LIN {X 0,Y 524.534,Z 584.102,A -85,B 0,C 180,E1 -4783.363,E2 -4783.363} C_VEL
LIN {X 0,Y 524.942,Z 571.861,A -85,B 0,C 180,E1 -4784.637,E2 -4784.637} C_VEL
LIN {X 0,Y 525.437,Z 560.491,A -85,B 0,C 180,E1 -4785.626,E2 -4785.626} C_VEL
LIN {X 0,Y 525.876,Z 547.102,A -85,B 0,C 180,E1 -4786.598,E2 -4786.598} C_VEL
LIN {X 0,Y 526.385,Z 533.833,A -85,B 0,C 180,E1 -4787.382,E2 -4787.382} C_VEL
LIN {X 0,Y 526.784,Z 519.311,A -85,B 0,C 180,E1 -4788.07,E2 -4788.07} C_VEL
LIN {X 0,Y 527.168,Z 504.263,A -85,B 0,C 180,E1 -4788.61,E2 -4788.61} C_VEL
LIN {X 0,Y 527.486,Z 489.588,A -85,B 0,C 180,E1 -4788.979,E2 -4788.979} C_VEL
LIN {X 0,Y 527.689,Z 461.99,A -85,B 0,C 180,E1 -4789.4,E2 -4789.4} C_VEL
LIN {X 0,Y 528.491,Z 335.003,A -85,B 0,C 180,E1 -4791.175,E2 -4791.175} C_VEL
LIN {X 0,Y 525.773,Z 320.948,A -85,B 0,C 180,E1 -4791.508,E2 -4791.508} C_VEL
LIN {X 0,Y 526.419,Z 300.055,A -85,B 0,C 180,E1 -4794.238,E2 -4794.238} C_VEL
LIN {X 0,Y 526.82,Z 285.888,A -85,B 0,C 180,E1 -4796.119,E2 -4796.119} C_VEL
LIN {X 0,Y 524.339,Z 274.589,A -85,B 0,C 180,E1 -4797.793,E2 -4797.793} C_VEL
LIN {X 0,Y 523.945,Z 272.841,A -85,B 0,C 180,E1 -4798.082,E2 -4798.082} C_VEL
LIN {X 0,Y 523.94,Z 272.844,A -85,B 0,C 180,E1 -4800.853,E2 -4800.853} C_VEL
LIN {X 0,Y 523.926,Z 272.849,A -85,B 0,C 180,E1 -4803.728,E2 -4803.728} C_VEL
LIN {X 0,Y 523.887,Z 272.856,A -85,B 0,C 180,E1 -4806.398,E2 -4806.398} C_VEL
LIN {X 0,Y 523.911,Z 272.847,A -85,B 0,C 180,E1 -4809.085,E2 -4809.085} C_VEL
LIN {X 0,Y 523.898,Z 272.854,A -85,B 0,C 180,E1 -4812.124,E2 -4812.124} C_VEL
LIN {X 0,Y 523.934,Z 272.843,A -85,B 0,C 180,E1 -4815.31,E2 -4815.31} C_VEL
LIN {X 0,Y 523.92,Z 272.846,A -85,B 0,C 180,E1 -4818.693,E2 -4818.693} C_VEL
LIN {X 0,Y 523.898,Z 272.853,A -85,B 0,C 180,E1 -4821.896,E2 -4821.896} C_VEL
LIN {X 0,Y 523.911,Z 272.843,A -85,B 0,C 180,E1 -4824.912,E2 -4824.912} C_VEL
LIN {X 0,Y 523.932,Z 272.847,A -85,B 0,C 180,E1 -4827.679,E2 -4827.679} C_VEL
LIN {X 0,Y 523.948,Z 272.84,A -85,B 0,C 180,E1 -4830.676,E2 -4830.676} C_VEL
LIN {X 0,Y 523.887,Z 272.854,A -85,B 0,C 180,E1 -4833.723,E2 -4833.723} C_VEL
LIN {X 0,Y 523.904,Z 272.848,A -85,B 0,C 180,E1 -4836.268,E2 -4836.268} C_VEL
LIN {X 0,Y 523.94,Z 272.842,A -85,B 0,C 180,E1 -4838.765,E2 -4838.765} C_VEL
LIN {X 0,Y 523.928,Z 272.844,A -85,B 0,C 180,E1 -4841.219,E2 -4841.219} C_VEL
LIN {X 0,Y 523.898,Z 272.855,A -85,B 0,C 180,E1 -4843.637,E2 -4843.637} C_VEL
LIN {X 0,Y 523.921,Z 272.84,A -85,B 0,C 180,E1 -4846.026,E2 -4846.026} C_VEL
LIN {X 0,Y 523.955,Z 272.834,A -85,B 0,C 180,E1 -4848.392,E2 -4848.392} C_VEL
LIN {X 0,Y 523.937,Z 272.848,A -85,B 0,C 180,E1 -4851.514,E2 -4851.514} C_VEL
LIN {X 0,Y 524.026,Z 272.827,A -85,B 0,C 180,E1 -4854.612,E2 -4854.612} C_VEL
LIN {X 0,Y 524.088,Z 272.823,A -85,B 0,C 180,E1 -4857.693,E2 -4857.693} C_VEL
LIN {X 0,Y 524.078,Z 272.826,A -85,B 0,C 180,E1 -4859.999,E2 -4859.999} C_VEL
LIN {X 0,Y 524.02,Z 272.834,A -85,B 0,C 180,E1 -4863.074,E2 -4863.074} C_VEL
LIN {X 0,Y 523.975,Z 272.827,A -85,B 0,C 180,E1 -4866.158,E2 -4866.158} C_VEL
LIN {X 0,Y 523.929,Z 272.844,A -85,B 0,C 180,E1 -4869.262,E2 -4869.262} C_VEL
LIN {X 0,Y 523.983,Z 272.84,A -85,B 0,C 180,E1 -4871.733,E2 -4871.733} C_VEL
LIN {X 0,Y 523.97,Z 272.838,A -85,B 0,C 180,E1 -4875.046,E2 -4875.046} C_VEL
LIN {X 0,Y 523.901,Z 272.841,A -85,B 0,C 180,E1 -4877.97,E2 -4877.97} C_VEL
LIN {X 0,Y 523.938,Z 272.84,A -85,B 0,C 180,E1 -4880.41,E2 -4880.41} C_VEL
LIN {X 0,Y 523.892,Z 272.85,A -85,B 0,C 180,E1 -4882.893,E2 -4882.893} C_VEL
LIN {X 0,Y 523.886,Z 272.847,A -85,B 0,C 180,E1 -4885.42,E2 -4885.42} C_VEL
LIN {X 0,Y 523.891,Z 272.841,A -85,B 0,C 180,E1 -4888.001,E2 -4888.001} C_VEL
LIN {X 0,Y 523.919,Z 272.846,A -85,B 0,C 180,E1 -4890.851,E2 -4890.851} C_VEL
LIN {X 0,Y 523.91,Z 272.844,A -85,B 0,C 180,E1 -4893.728,E2 -4893.728} C_VEL
LIN {X 0,Y 523.881,Z 272.841,A -85,B 0,C 180,E1 -4896.399,E2 -4896.399} C_VEL
LIN {X 0,Y 523.903,Z 272.85,A -85,B 0,C 180,E1 -4899.084,E2 -4899.084} C_VEL
LIN {X 0,Y 523.894,Z 272.847,A -85,B 0,C 180,E1 -4902.122,E2 -4902.122} C_VEL
LIN {X 0,Y 523.921,Z 272.843,A -85,B 0,C 180,E1 -4905.31,E2 -4905.31} C_VEL
LIN {X 0,Y 523.874,Z 272.85,A -85,B 0,C 180,E1 -4906.857,E2 -4906.857} C_VEL
LIN {X 0,Y 523.204,Z 272.935,A -85,B 0,C 180,E1 -4907.499,E2 -4907.499} C_VEL
LIN {X 0,Y 520.347,Z 273.291,A -85,B 0,C 180,E1 -4908.541,E2 -4908.541} C_VEL
LIN {X 0,Y 517.946,Z 273.592,A -85,B 0,C 180,E1 -4909.38,E2 -4909.38} C_VEL
LIN {X 0,Y 516.935,Z 273.715,A -85,B 0,C 180,E1 -4910.028,E2 -4910.028} C_VEL
LIN {X 0,Y 516.863,Z 273.724,A -85,B 0,C 180,E1 -4910.247,E2 -4910.247} C_VEL
LIN {X 0,Y 516.859,Z 273.723,A -85,B 0,C 180,E1 -4913.342,E2 -4913.342} C_VEL
LIN {X 0,Y 516.869,Z 273.723,A -85,B 0,C 180,E1 -4916.118,E2 -4916.118} C_VEL
LIN {X 0,Y 516.871,Z 273.724,A -85,B 0,C 180,E1 -4918.935,E2 -4918.935} C_VEL
LIN {X 0,Y 516.891,Z 273.72,A -85,B 0,C 180,E1 -4921.583,E2 -4921.583} C_VEL
LIN {X 0,Y 516.908,Z 273.717,A -85,B 0,C 180,E1 -4924.21,E2 -4924.21} C_VEL
LIN {X 0,Y 516.841,Z 273.733,A -85,B 0,C 180,E1 -4926.775,E2 -4926.775} C_VEL
LIN {X 0,Y 516.92,Z 273.713,A -85,B 0,C 180,E1 -4929.731,E2 -4929.731} C_VEL
LIN {X 0,Y 516.902,Z 273.726,A -85,B 0,C 180,E1 -4932.595,E2 -4932.595} C_VEL
LIN {X 0,Y 516.923,Z 273.72,A -85,B 0,C 180,E1 -4935.03,E2 -4935.03} C_VEL
LIN {X 0,Y 516.986,Z 273.711,A -85,B 0,C 180,E1 -4938.234,E2 -4938.234} C_VEL
LIN {X 0,Y 516.947,Z 273.713,A -85,B 0,C 180,E1 -4941.399,E2 -4941.399} C_VEL
LIN {X 0,Y 516.983,Z 273.709,A -85,B 0,C 180,E1 -4943.756,E2 -4943.756} C_VEL
LIN {X 0,Y 516.996,Z 273.713,A -85,B 0,C 180,E1 -4946.883,E2 -4946.883} C_VEL
LIN {X 0,Y 517.061,Z 273.704,A -85,B 0,C 180,E1 -4950,E2 -4950} C_VEL
LIN {X 0,Y 516.997,Z 273.713,A -85,B 0,C 180,E1 -4953.117,E2 -4953.117} C_VEL
LIN {X 0,Y 516.965,Z 273.73,A -85,B 0,C 180,E1 -4954.971,E2 -4954.971} C_VEL
LIN {X 0,Y 519.171,Z 284.58,A -85,B 0,C 180,E1 -4956.802,E2 -4956.802} C_VEL
LIN {X 0,Y 518.896,Z 293.997,A -85,B 0,C 180,E1 -4958.262,E2 -4958.262} C_VEL
LIN {X 0,Y 521.949,Z 308.526,A -85,B 0,C 180,E1 -4958.616,E2 -4958.616} C_VEL
LIN {X 0,Y 520.88,Z 458.501,A -85,B 0,C 180,E1 -4960.765,E2 -4960.765} C_VEL
LIN {X 0,Y 520.579,Z 474.054,A -85,B 0,C 180,E1 -4961.14,E2 -4961.14} C_VEL
LIN {X 0,Y 520.181,Z 488.457,A -85,B 0,C 180,E1 -4961.643,E2 -4961.643} C_VEL
LIN {X 0,Y 519.746,Z 502.613,A -85,B 0,C 180,E1 -4962.296,E2 -4962.296} C_VEL
LIN {X 0,Y 519.223,Z 517.187,A -85,B 0,C 180,E1 -4963.151,E2 -4963.151} C_VEL
LIN {X 0,Y 518.677,Z 530.47,A -85,B 0,C 180,E1 -4964.116,E2 -4964.116} C_VEL
LIN {X 0,Y 518.171,Z 543.252,A -85,B 0,C 180,E1 -4965.246,E2 -4965.246} C_VEL
LIN {X 0,Y 517.693,Z 553.804,A -85,B 0,C 180,E1 -4966.361,E2 -4966.361} C_VEL
LIN {X 0,Y 517.267,Z 564.356,A -85,B 0,C 180,E1 -4967.687,E2 -4967.687} C_VEL
LIN {X 0,Y 516.921,Z 573.373,A -85,B 0,C 180,E1 -4969.044,E2 -4969.044} C_VEL
LIN {X 0,Y 516.665,Z 581.006,A -85,B 0,C 180,E1 -4970.419,E2 -4970.419} C_VEL
LIN {X 0,Y 516.487,Z 587.844,A -85,B 0,C 180,E1 -4971.916,E2 -4971.916} C_VEL
LIN {X 0,Y 516.396,Z 592.797,A -85,B 0,C 180,E1 -4973.245,E2 -4973.245} C_VEL
LIN {X 0,Y 516.314,Z 597.706,A -85,B 0,C 180,E1 -4974.958,E2 -4974.958} C_VEL
LIN {X 0,Y 516.195,Z 601.163,A -85,B 0,C 180,E1 -4976.697,E2 -4976.697} C_VEL
LIN {X 0,Y 516.159,Z 603.183,A -85,B 0,C 180,E1 -4978.46,E2 -4978.46} C_VEL
LIN {X 0,Y 516.178,Z 603.657,A -85,B 0,C 180,E1 -4979.384,E2 -4979.384} C_VEL
LIN {X 0,Y 516.169,Z 603.47,A -85,B 0,C 180,E1 -4981.157,E2 -4981.157} C_VEL
LIN {X 0,Y 516.161,Z 602.457,A -85,B 0,C 180,E1 -4982.419,E2 -4982.419} C_VEL
LIN {X 0,Y 516.204,Z 600.239,A -85,B 0,C 180,E1 -4983.931,E2 -4983.931} C_VEL
LIN {X 0,Y 516.239,Z 597.469,A -85,B 0,C 180,E1 -4985.235,E2 -4985.235} C_VEL
LIN {X 0,Y 516.374,Z 592.998,A -85,B 0,C 180,E1 -4986.786,E2 -4986.786} C_VEL
LIN {X 0,Y 516.523,Z 587.426,A -85,B 0,C 180,E1 -4988.282,E2 -4988.282} C_VEL
LIN {X 0,Y 516.714,Z 580.712,A -85,B 0,C 180,E1 -4989.735,E2 -4989.735} C_VEL
LIN {X 0,Y 516.974,Z 572.603,A -85,B 0,C 180,E1 -4991.179,E2 -4991.179} C_VEL
LIN {X 0,Y 517.262,Z 563.509,A -85,B 0,C 180,E1 -4992.526,E2 -4992.526} C_VEL
LIN {X 0,Y 517.757,Z 553.155,A -85,B 0,C 180,E1 -4993.808,E2 -4993.808} C_VEL
LIN {X 0,Y 518.201,Z 542.018,A -85,B 0,C 180,E1 -4994.968,E2 -4994.968} C_VEL
LIN {X 0,Y 518.741,Z 528.872,A -85,B 0,C 180,E1 -4996.104,E2 -4996.104} C_VEL
LIN {X 0,Y 519.295,Z 515.044,A -85,B 0,C 180,E1 -4997.081,E2 -4997.081} C_VEL
LIN {X 0,Y 519.785,Z 501.397,A -85,B 0,C 180,E1 -4997.859,E2 -4997.859} C_VEL
LIN {X 0,Y 520.233,Z 487.144,A -85,B 0,C 180,E1 -4998.5,E2 -4998.5} C_VEL
LIN {X 0,Y 520.632,Z 472.824,A -85,B 0,C 180,E1 -4998.985,E2 -4998.985} C_VEL
LIN {X 0,Y 520.874,Z 457.657,A -85,B 0,C 180,E1 -4999.342,E2 -4999.342} C_VEL
LIN {X 0,Y 521.954,Z 307.911,A -85,B 0,C 180,E1 -5001.486,E2 -5001.486} C_VEL
LIN {X 0,Y 518.89,Z 294.114,A -85,B 0,C 180,E1 -5001.847,E2 -5001.847} C_VEL
LIN {X 0,Y 519.152,Z 284.912,A -85,B 0,C 180,E1 -5003.278,E2 -5003.278} C_VEL
LIN {X 0,Y 517.737,Z 277.455,A -85,B 0,C 180,E1 -5004.532,E2 -5004.532} C_VEL
LIN {X 0,Y 516.899,Z 273.725,A -85,B 0,C 180,E1 -5005.179,E2 -5005.179} C_VEL
LIN {X 0,Y 516.866,Z 273.728,A -85,B 0,C 180,E1 -5007.977,E2 -5007.977} C_VEL
LIN {X 0,Y 516.918,Z 273.72,A -85,B 0,C 180,E1 -5010.697,E2 -5010.697} C_VEL
LIN {X 0,Y 516.928,Z 273.72,A -85,B 0,C 180,E1 -5013.804,E2 -5013.804} C_VEL
LIN {X 0,Y 516.856,Z 273.728,A -85,B 0,C 180,E1 -5016.778,E2 -5016.778} C_VEL
LIN {X 0,Y 516.923,Z 273.72,A -85,B 0,C 180,E1 -5019.732,E2 -5019.732} C_VEL
LIN {X 0,Y 516.916,Z 273.719,A -85,B 0,C 180,E1 -5022.597,E2 -5022.597} C_VEL
LIN {X 0,Y 516.926,Z 273.723,A -85,B 0,C 180,E1 -5025.031,E2 -5025.031} C_VEL
LIN {X 0,Y 516.951,Z 273.713,A -85,B 0,C 180,E1 -5028.235,E2 -5028.235} C_VEL
LIN {X 0,Y 516.951,Z 273.716,A -85,B 0,C 180,E1 -5031.401,E2 -5031.401} C_VEL
LIN {X 0,Y 516.988,Z 273.707,A -85,B 0,C 180,E1 -5033.758,E2 -5033.758} C_VEL
LIN {X 0,Y 517,Z 273.712,A -85,B 0,C 180,E1 -5036.884,E2 -5036.884} C_VEL
LIN {X 0,Y 517.067,Z 273.697,A -85,B 0,C 180,E1 -5040.001,E2 -5040.001} C_VEL
LIN {X 0,Y 516.997,Z 273.712,A -85,B 0,C 180,E1 -5043.118,E2 -5043.118} C_VEL
LIN {X 0,Y 516.974,Z 273.711,A -85,B 0,C 180,E1 -5046.245,E2 -5046.245} C_VEL
LIN {X 0,Y 516.929,Z 273.716,A -85,B 0,C 180,E1 -5049.391,E2 -5049.391} C_VEL
LIN {X 0,Y 516.941,Z 273.713,A -85,B 0,C 180,E1 -5051.808,E2 -5051.808} C_VEL
LIN {X 0,Y 516.934,Z 273.717,A -85,B 0,C 180,E1 -5055.147,E2 -5055.147} C_VEL
LIN {X 0,Y 516.906,Z 273.72,A -85,B 0,C 180,E1 -5058.224,E2 -5058.224} C_VEL
LIN {X 0,Y 516.902,Z 273.725,A -85,B 0,C 180,E1 -5060.703,E2 -5060.703} C_VEL
LIN {X 0,Y 516.875,Z 273.723,A -85,B 0,C 180,E1 -5064.075,E2 -5064.075} C_VEL
LIN {X 0,Y 516.827,Z 273.733,A -85,B 0,C 180,E1 -5066.664,E2 -5066.664} C_VEL
LIN {X 0,Y 516.889,Z 273.719,A -85,B 0,C 180,E1 -5069.522,E2 -5069.522} C_VEL
LIN {X 0,Y 516.883,Z 273.726,A -85,B 0,C 180,E1 -5072.544,E2 -5072.544} C_VEL
LIN {X 0,Y 516.841,Z 273.725,A -85,B 0,C 180,E1 -5075.328,E2 -5075.328} C_VEL
LIN {X 0,Y 516.861,Z 273.724,A -85,B 0,C 180,E1 -5078.718,E2 -5078.718} C_VEL
LIN {X 0,Y 516.832,Z 273.73,A -85,B 0,C 180,E1 -5081.784,E2 -5081.784} C_VEL
LIN {X 0,Y 516.891,Z 273.72,A -85,B 0,C 180,E1 -5085.008,E2 -5085.008} C_VEL
LIN {X 0,Y 516.847,Z 273.729,A -85,B 0,C 180,E1 -5088.408,E2 -5088.408} C_VEL
LIN {X 0,Y 516.869,Z 273.724,A -85,B 0,C 180,E1 -5091.284,E2 -5091.284} C_VEL
LIN {X 0,Y 516.849,Z 273.727,A -85,B 0,C 180,E1 -5094.674,E2 -5094.674} C_VEL
LIN {X 0,Y 516.892,Z 273.724,A -85,B 0,C 180,E1 -5097.458,E2 -5097.458} C_VEL
LIN {X 0,Y 516.919,Z 273.721,A -85,B 0,C 180,E1 -5100.696,E2 -5100.696} C_VEL
LIN {X 0,Y 516.931,Z 273.784,A -85,B 0,C 180,E1 -5101.727,E2 -5101.727} C_VEL
LIN {X 0,Y 519.927,Z 287.034,A -85,B 0,C 180,E1 -5103.725,E2 -5103.725} C_VEL
LIN {X 0,Y 519.499,Z 301.184,A -85,B 0,C 180,E1 -5105.632,E2 -5105.632} C_VEL
LIN {X 0,Y 518.899,Z 320.095,A -85,B 0,C 180,E1 -5108.134,E2 -5108.134} C_VEL
LIN {X 0,Y 518.881,Z 320.674,A -85,B 0,C 180,E1 -5108.209,E2 -5108.209} C_VEL
LIN {X 0,Y 521.85,Z 335.907,A -85,B 0,C 180,E1 -5108.561,E2 -5108.561} C_VEL
LIN {X 0,Y 520.802,Z 487.578,A -85,B 0,C 180,E1 -5110.736,E2 -5110.736} C_VEL
LIN {X 0,Y 520.438,Z 503.039,A -85,B 0,C 180,E1 -5111.115,E2 -5111.115} C_VEL
LIN {X 0,Y 520.079,Z 517.761,A -85,B 0,C 180,E1 -5111.638,E2 -5111.638} C_VEL
LIN {X 0,Y 519.572,Z 531.624,A -85,B 0,C 180,E1 -5112.282,E2 -5112.282} C_VEL
LIN {X 0,Y 519.061,Z 545.223,A -85,B 0,C 180,E1 -5113.077,E2 -5113.077} C_VEL
LIN {X 0,Y 518.552,Z 559.058,A -85,B 0,C 180,E1 -5114.072,E2 -5114.072} C_VEL
LIN {X 0,Y 518.007,Z 571.561,A -85,B 0,C 180,E1 -5115.163,E2 -5115.163} C_VEL
LIN {X 0,Y 517.537,Z 583.83,A -85,B 0,C 180,E1 -5116.453,E2 -5116.453} C_VEL
LIN {X 0,Y 517.106,Z 594.731,A -85,B 0,C 180,E1 -5117.84,E2 -5117.84} C_VEL
LIN {X 0,Y 516.883,Z 603.805,A -85,B 0,C 180,E1 -5119.225,E2 -5119.225} C_VEL
LIN {X 0,Y 516.598,Z 611.326,A -85,B 0,C 180,E1 -5120.605,E2 -5120.605} C_VEL
LIN {X 0,Y 516.452,Z 618.347,A -85,B 0,C 180,E1 -5122.179,E2 -5122.179} C_VEL
LIN {X 0,Y 516.329,Z 623.863,A -85,B 0,C 180,E1 -5123.749,E2 -5123.749} C_VEL
LIN {X 0,Y 516.238,Z 628.034,A -85,B 0,C 180,E1 -5125.315,E2 -5125.315} C_VEL
LIN {X 0,Y 516.272,Z 630.959,A -85,B 0,C 180,E1 -5126.879,E2 -5126.879} C_VEL
LIN {X 0,Y 516.19,Z 632.701,A -85,B 0,C 180,E1 -5128.44,E2 -5128.44} C_VEL
LIN {X 0,Y 516.151,Z 633.299,A -85,B 0,C 180,E1 -5130,E2 -5130} C_VEL
LIN {X 0,Y 516.19,Z 632.7,A -85,B 0,C 180,E1 -5131.561,E2 -5131.561} C_VEL
LIN {X 0,Y 516.272,Z 630.958,A -85,B 0,C 180,E1 -5133.122,E2 -5133.122} C_VEL
LIN {X 0,Y 516.239,Z 628.038,A -85,B 0,C 180,E1 -5134.686,E2 -5134.686} C_VEL
LIN {X 0,Y 516.329,Z 623.878,A -85,B 0,C 180,E1 -5136.252,E2 -5136.252} C_VEL
LIN {X 0,Y 516.452,Z 618.362,A -85,B 0,C 180,E1 -5137.821,E2 -5137.821} C_VEL
LIN {X 0,Y 516.609,Z 611.34,A -85,B 0,C 180,E1 -5139.396,E2 -5139.396} C_VEL
LIN {X 0,Y 516.882,Z 603.828,A -85,B 0,C 180,E1 -5140.775,E2 -5140.775} C_VEL
LIN {X 0,Y 517.115,Z 595.04,A -85,B 0,C 180,E1 -5142.121,E2 -5142.121} C_VEL
LIN {X 0,Y 517.502,Z 585.521,A -85,B 0,C 180,E1 -5143.348,E2 -5143.348} C_VEL
LIN {X 0,Y 517.861,Z 574.624,A -85,B 0,C 180,E1 -5144.541,E2 -5144.541} C_VEL
LIN {X 0,Y 518.401,Z 563.326,A -85,B 0,C 180,E1 -5145.581,E2 -5145.581} C_VEL
LIN {X 0,Y 518.878,Z 549.722,A -85,B 0,C 180,E1 -5146.626,E2 -5146.626} C_VEL
LIN {X 0,Y 519.501,Z 535.348,A -85,B 0,C 180,E1 -5147.518,E2 -5147.518} C_VEL
LIN {X 0,Y 519.929,Z 521.3,A -85,B 0,C 180,E1 -5148.215,E2 -5148.215} C_VEL
LIN {X 0,Y 520.365,Z 506.255,A -85,B 0,C 180,E1 -5148.786,E2 -5148.786} C_VEL
LIN {X 0,Y 520.725,Z 490.844,A -85,B 0,C 180,E1 -5149.199,E2 -5149.199} C_VEL
LIN {X 0,Y 520.937,Z 469.871,A -85,B 0,C 180,E1 -5149.542,E2 -5149.542} C_VEL
LIN {X 0,Y 521.864,Z 335.914,A -85,B 0,C 180,E1 -5151.441,E2 -5151.441} C_VEL
LIN {X 0,Y 518.892,Z 320.749,A -85,B 0,C 180,E1 -5151.808,E2 -5151.808} C_VEL
LIN {X 0,Y 519.558,Z 301.452,A -85,B 0,C 180,E1 -5154.366,E2 -5154.366} C_VEL
LIN {X 0,Y 519.978,Z 287.3,A -85,B 0,C 180,E1 -5156.273,E2 -5156.273} C_VEL
LIN {X 0,Y 516.903,Z 273.72,A -85,B 0,C 180,E1 -5158.346,E2 -5158.346} C_VEL
LIN {X 0,Y 516.889,Z 273.722,A -85,B 0,C 180,E1 -5161.109,E2 -5161.109} C_VEL
LIN {X 0,Y 516.881,Z 273.728,A -85,B 0,C 180,E1 -5163.961,E2 -5163.961} C_VEL
LIN {X 0,Y 516.843,Z 273.73,A -85,B 0,C 180,E1 -5166.748,E2 -5166.748} C_VEL
LIN {X 0,Y 516.857,Z 273.729,A -85,B 0,C 180,E1 -5169.723,E2 -5169.723} C_VEL
LIN {X 0,Y 516.841,Z 273.725,A -85,B 0,C 180,E1 -5172.835,E2 -5172.835} C_VEL
LIN {X 0,Y 516.895,Z 273.72,A -85,B 0,C 180,E1 -5175.006,E2 -5175.006} C_VEL
LIN {X 0,Y 516.885,Z 273.725,A -85,B 0,C 180,E1 -5178.401,E2 -5178.401} C_VEL
LIN {X 0,Y 516.87,Z 273.721,A -85,B 0,C 180,E1 -5181.282,E2 -5181.282} C_VEL
LIN {X 0,Y 516.847,Z 273.723,A -85,B 0,C 180,E1 -5184.672,E2 -5184.672} C_VEL
LIN {X 0,Y 516.891,Z 273.721,A -85,B 0,C 180,E1 -5187.456,E2 -5187.456} C_VEL
LIN {X 0,Y 516.916,Z 273.717,A -85,B 0,C 180,E1 -5190.694,E2 -5190.694} C_VEL
LIN {X 0,Y 516.864,Z 273.731,A -85,B 0,C 180,E1 -5193.82,E2 -5193.82} C_VEL
LIN {X 0,Y 516.853,Z 273.724,A -85,B 0,C 180,E1 -5196.775,E2 -5196.775} C_VEL
LIN {X 0,Y 516.935,Z 273.722,A -85,B 0,C 180,E1 -5199.731,E2 -5199.731} C_VEL
LIN {X 0,Y 516.879,Z 273.722,A -85,B 0,C 180,E1 -5202.593,E2 -5202.593} C_VEL
LIN {X 0,Y 516.937,Z 273.713,A -85,B 0,C 180,E1 -5205.029,E2 -5205.029} C_VEL
LIN {X 0,Y 516.919,Z 273.711,A -85,B 0,C 180,E1 -5208.232,E2 -5208.232} C_VEL
LIN {X 0,Y 516.911,Z 273.721,A -85,B 0,C 180,E1 -5211.398,E2 -5211.398} C_VEL
LIN {X 0,Y 516.976,Z 273.705,A -85,B 0,C 180,E1 -5214.538,E2 -5214.538} C_VEL
LIN {X 0,Y 517.059,Z 273.698,A -85,B 0,C 180,E1 -5217.662,E2 -5217.662} C_VEL
LIN {X 0,Y 517.048,Z 273.702,A -85,B 0,C 180,E1 -5219.999,E2 -5219.999} C_VEL
LIN {X 0,Y 517.059,Z 273.698,A -85,B 0,C 180,E1 -5222.336,E2 -5222.336} C_VEL
LIN {X 0,Y 516.965,Z 273.708,A -85,B 0,C 180,E1 -5225.459,E2 -5225.459} C_VEL
LIN {X 0,Y 516.905,Z 273.712,A -85,B 0,C 180,E1 -5228.6,E2 -5228.6} C_VEL
LIN {X 0,Y 516.942,Z 273.716,A -85,B 0,C 180,E1 -5231.806,E2 -5231.806} C_VEL
LIN {X 0,Y 516.923,Z 273.717,A -85,B 0,C 180,E1 -5235.141,E2 -5235.141} C_VEL
LIN {X 0,Y 516.863,Z 273.716,A -85,B 0,C 180,E1 -5238.223,E2 -5238.223} C_VEL
LIN {X 0,Y 516.888,Z 273.719,A -85,B 0,C 180,E1 -5240.701,E2 -5240.701} C_VEL
LIN {X 0,Y 516.842,Z 273.733,A -85,B 0,C 180,E1 -5243.223,E2 -5243.223} C_VEL
LIN {X 0,Y 516.867,Z 273.714,A -85,B 0,C 180,E1 -5246.181,E2 -5246.181} C_VEL
LIN {X 0,Y 516.888,Z 273.723,A -85,B 0,C 180,E1 -5249.305,E2 -5249.305} C_VEL
LIN {X 0,Y 516.879,Z 273.722,A -85,B 0,C 180,E1 -5252.542,E2 -5252.542} C_VEL
LIN {X 0,Y 516.844,Z 273.723,A -85,B 0,C 180,E1 -5255.327,E2 -5255.327} C_VEL
LIN {X 0,Y 516.862,Z 273.718,A -85,B 0,C 180,E1 -5257.941,E2 -5257.941} C_VEL
LIN {X 0,Y 516.845,Z 273.728,A -85,B 0,C 180,E1 -5260.743,E2 -5260.743} C_VEL
LIN {X 0,Y 516.865,Z 273.719,A -85,B 0,C 180,E1 -5263.902,E2 -5263.902} C_VEL
LIN {X 0,Y 516.827,Z 273.728,A -85,B 0,C 180,E1 -5266.858,E2 -5266.858} C_VEL
LIN {X 0,Y 516.866,Z 273.724,A -85,B 0,C 180,E1 -5269.589,E2 -5269.589} C_VEL
LIN {X 0,Y 516.863,Z 273.724,A -85,B 0,C 180,E1 -5270.247,E2 -5270.247} C_VEL
LIN {X 0,Y 516.225,Z 273.81,A -85,B 0,C 180,E1 -5270.897,E2 -5270.897} C_VEL
LIN {X 0,Y 513.383,Z 274.161,A -85,B 0,C 180,E1 -5271.952,E2 -5271.952} C_VEL
LIN {X 0,Y 510.954,Z 274.461,A -85,B 0,C 180,E1 -5272.802,E2 -5272.802} C_VEL
LIN {X 0,Y 509.898,Z 274.59,A -85,B 0,C 180,E1 -5273.459,E2 -5273.459} C_VEL
LIN {X 0,Y 509.805,Z 274.599,A -85,B 0,C 180,E1 -5273.681,E2 -5273.681} C_VEL
LIN {X 0,Y 509.825,Z 274.603,A -85,B 0,C 180,E1 -5276.537,E2 -5276.537} C_VEL
LIN {X 0,Y 509.824,Z 274.597,A -85,B 0,C 180,E1 -5279.333,E2 -5279.333} C_VEL
LIN {X 0,Y 509.866,Z 274.594,A -85,B 0,C 180,E1 -5282.053,E2 -5282.053} C_VEL
LIN {X 0,Y 509.819,Z 274.604,A -85,B 0,C 180,E1 -5284.701,E2 -5284.701} C_VEL
LIN {X 0,Y 509.807,Z 274.604,A -85,B 0,C 180,E1 -5287.457,E2 -5287.457} C_VEL
LIN {X 0,Y 509.898,Z 274.588,A -85,B 0,C 180,E1 -5289.844,E2 -5289.844} C_VEL
LIN {X 0,Y 509.862,Z 274.596,A -85,B 0,C 180,E1 -5293.174,E2 -5293.174} C_VEL
LIN {X 0,Y 509.843,Z 274.597,A -85,B 0,C 180,E1 -5295.634,E2 -5295.634} C_VEL
LIN {X 0,Y 509.912,Z 274.593,A -85,B 0,C 180,E1 -5298.874,E2 -5298.874} C_VEL
LIN {X 0,Y 509.931,Z 274.588,A -85,B 0,C 180,E1 -5302.078,E2 -5302.078} C_VEL
LIN {X 0,Y 509.96,Z 274.589,A -85,B 0,C 180,E1 -5304.464,E2 -5304.464} C_VEL
LIN {X 0,Y 510.033,Z 274.576,A -85,B 0,C 180,E1 -5307.631,E2 -5307.631} C_VEL
LIN {X 0,Y 510.032,Z 274.58,A -85,B 0,C 180,E1 -5310,E2 -5310} C_VEL
LIN {X 0,Y 510.034,Z 274.583,A -85,B 0,C 180,E1 -5312.369,E2 -5312.369} C_VEL
LIN {X 0,Y 509.92,Z 274.769,A -85,B 0,C 180,E1 -5314.743,E2 -5314.743} C_VEL
LIN {X 0,Y 512.323,Z 286.141,A -85,B 0,C 180,E1 -5316.696,E2 -5316.696} C_VEL
LIN {X 0,Y 512.099,Z 294.418,A -85,B 0,C 180,E1 -5317.967,E2 -5317.967} C_VEL
LIN {X 0,Y 515.357,Z 309.658,A -85,B 0,C 180,E1 -5318.342,E2 -5318.342} C_VEL
LIN {X 0,Y 514.197,Z 458.728,A -85,B 0,C 180,E1 -5320.508,E2 -5320.508} C_VEL
LIN {X 0,Y 513.853,Z 474.322,A -85,B 0,C 180,E1 -5320.889,E2 -5320.889} C_VEL
LIN {X 0,Y 513.396,Z 489.938,A -85,B 0,C 180,E1 -5321.448,E2 -5321.448} C_VEL
LIN {X 0,Y 512.93,Z 504.732,A -85,B 0,C 180,E1 -5322.161,E2 -5322.161} C_VEL
LIN {X 0,Y 512.354,Z 518.973,A -85,B 0,C 180,E1 -5323.029,E2 -5323.029} C_VEL
LIN {X 0,Y 511.777,Z 531.972,A -85,B 0,C 180,E1 -5324.006,E2 -5324.006} C_VEL
LIN {X 0,Y 511.218,Z 544.434,A -85,B 0,C 180,E1 -5325.141,E2 -5325.141} C_VEL
LIN {X 0,Y 510.694,Z 555.814,A -85,B 0,C 180,E1 -5326.386,E2 -5326.386} C_VEL
LIN {X 0,Y 510.269,Z 565.415,A -85,B 0,C 180,E1 -5327.638,E2 -5327.638} C_VEL
LIN {X 0,Y 509.876,Z 574.856,A -85,B 0,C 180,E1 -5329.108,E2 -5329.108} C_VEL
LIN {X 0,Y 509.598,Z 582.882,A -85,B 0,C 180,E1 -5330.629,E2 -5330.629} C_VEL
LIN {X 0,Y 509.394,Z 589.389,A -85,B 0,C 180,E1 -5332.145,E2 -5332.145} C_VEL
LIN {X 0,Y 509.282,Z 594.35,A -85,B 0,C 180,E1 -5333.589,E2 -5333.589} C_VEL
LIN {X 0,Y 509.178,Z 598.891,A -85,B 0,C 180,E1 -5335.332,E2 -5335.332} C_VEL
LIN {X 0,Y 509.072,Z 601.992,A -85,B 0,C 180,E1 -5337.101,E2 -5337.101} C_VEL
LIN {X 0,Y 509.069,Z 603.656,A -85,B 0,C 180,E1 -5338.893,E2 -5338.893} C_VEL
LIN {X 0,Y 509.073,Z 603.861,A -85,B 0,C 180,E1 -5340.716,E2 -5340.716} C_VEL
LIN {X 0,Y 509.063,Z 603.397,A -85,B 0,C 180,E1 -5341.641,E2 -5341.641} C_VEL
LIN {X 0,Y 509.065,Z 602.476,A -85,B 0,C 180,E1 -5342.636,E2 -5342.636} C_VEL
LIN {X 0,Y 509.11,Z 600.269,A -85,B 0,C 180,E1 -5344.083,E2 -5344.083} C_VEL
LIN {X 0,Y 509.253,Z 596.09,A -85,B 0,C 180,E1 -5345.909,E2 -5345.909} C_VEL
LIN {X 0,Y 509.343,Z 591.484,A -85,B 0,C 180,E1 -5347.38,E2 -5347.38} C_VEL
LIN {X 0,Y 509.499,Z 585.594,A -85,B 0,C 180,E1 -5348.874,E2 -5348.874} C_VEL
LIN {X 0,Y 509.761,Z 578.213,A -85,B 0,C 180,E1 -5350.388,E2 -5350.388} C_VEL
LIN {X 0,Y 510.082,Z 569.035,A -85,B 0,C 180,E1 -5351.928,E2 -5351.928} C_VEL
LIN {X 0,Y 510.526,Z 559.294,A -85,B 0,C 180,E1 -5353.28,E2 -5353.28} C_VEL
LIN {X 0,Y 510.988,Z 548.454,A -85,B 0,C 180,E1 -5354.541,E2 -5354.541} C_VEL
LIN {X 0,Y 511.593,Z 536.171,A -85,B 0,C 180,E1 -5355.729,E2 -5355.729} C_VEL
LIN {X 0,Y 512.184,Z 522.977,A -85,B 0,C 180,E1 -5356.783,E2 -5356.783} C_VEL
LIN {X 0,Y 512.733,Z 509.369,A -85,B 0,C 180,E1 -5357.671,E2 -5357.671} C_VEL
LIN {X 0,Y 513.22,Z 496.025,A -85,B 0,C 180,E1 -5358.374,E2 -5358.374} C_VEL
LIN {X 0,Y 513.66,Z 480.653,A -85,B 0,C 180,E1 -5358.998,E2 -5358.998} C_VEL
LIN {X 0,Y 514.075,Z 464.869,A -85,B 0,C 180,E1 -5359.451,E2 -5359.451} C_VEL
LIN {X 0,Y 514.305,Z 448.138,A -85,B 0,C 180,E1 -5359.752,E2 -5359.752} C_VEL
LIN {X 0,Y 515.359,Z 309.335,A -85,B 0,C 180,E1 -5361.756,E2 -5361.756} C_VEL
LIN {X 0,Y 512.069,Z 294.496,A -85,B 0,C 180,E1 -5362.13,E2 -5362.13} C_VEL
LIN {X 0,Y 512.31,Z 286.641,A -85,B 0,C 180,E1 -5363.365,E2 -5363.365} C_VEL
LIN {X 0,Y 510.786,Z 278.831,A -85,B 0,C 180,E1 -5364.7,E2 -5364.7} C_VEL
LIN {X 0,Y 509.868,Z 274.602,A -85,B 0,C 180,E1 -5365.47,E2 -5365.47} C_VEL
LIN {X 0,Y 509.809,Z 274.605,A -85,B 0,C 180,E1 -5368.411,E2 -5368.411} C_VEL
LIN {X 0,Y 509.868,Z 274.601,A -85,B 0,C 180,E1 -5371.157,E2 -5371.157} C_VEL
LIN {X 0,Y 509.894,Z 274.596,A -85,B 0,C 180,E1 -5373.83,E2 -5373.83} C_VEL
LIN {X 0,Y 509.82,Z 274.603,A -85,B 0,C 180,E1 -5376.438,E2 -5376.438} C_VEL
LIN {X 0,Y 509.901,Z 274.593,A -85,B 0,C 180,E1 -5379.846,E2 -5379.846} C_VEL
LIN {X 0,Y 509.872,Z 274.602,A -85,B 0,C 180,E1 -5383.176,E2 -5383.176} C_VEL
LIN {X 0,Y 509.849,Z 274.6,A -85,B 0,C 180,E1 -5385.635,E2 -5385.635} C_VEL
LIN {X 0,Y 509.898,Z 274.596,A -85,B 0,C 180,E1 -5388.876,E2 -5388.876} C_VEL
LIN {X 0,Y 509.936,Z 274.586,A -85,B 0,C 180,E1 -5392.08,E2 -5392.08} C_VEL
LIN {X 0,Y 509.965,Z 274.583,A -85,B 0,C 180,E1 -5394.466,E2 -5394.466} C_VEL
LIN {X 0,Y 510.038,Z 274.575,A -85,B 0,C 180,E1 -5397.632,E2 -5397.632} C_VEL
LIN {X 0,Y 510.053,Z 274.578,A -85,B 0,C 180,E1 -5400.791,E2 -5400.791} C_VEL
LIN {X 0,Y 509.938,Z 274.59,A -85,B 0,C 180,E1 -5403.161,E2 -5403.161} C_VEL
LIN {X 0,Y 509.928,Z 274.589,A -85,B 0,C 180,E1 -5406.331,E2 -5406.331} C_VEL
LIN {X 0,Y 509.89,Z 274.597,A -85,B 0,C 180,E1 -5408.722,E2 -5408.722} C_VEL
LIN {X 0,Y 509.894,Z 274.591,A -85,B 0,C 180,E1 -5411.933,E2 -5411.933} C_VEL
LIN {X 0,Y 509.884,Z 274.594,A -85,B 0,C 180,E1 -5415.243,E2 -5415.243} C_VEL
LIN {X 0,Y 509.851,Z 274.603,A -85,B 0,C 180,E1 -5418.485,E2 -5418.485} C_VEL
LIN {X 0,Y 509.84,Z 274.601,A -85,B 0,C 180,E1 -5421.003,E2 -5421.003} C_VEL
LIN {X 0,Y 509.809,Z 274.6,A -85,B 0,C 180,E1 -5423.565,E2 -5423.565} C_VEL
LIN {X 0,Y 509.798,Z 274.608,A -85,B 0,C 180,E1 -5426.356,E2 -5426.356} C_VEL
LIN {X 0,Y 509.84,Z 274.599,A -85,B 0,C 180,E1 -5428.847,E2 -5428.847} C_VEL
LIN {X 0,Y 509.802,Z 274.601,A -85,B 0,C 180,E1 -5431.592,E2 -5431.592} C_VEL
LIN {X 0,Y 509.825,Z 274.605,A -85,B 0,C 180,E1 -5434.416,E2 -5434.416} C_VEL
LIN {X 0,Y 509.771,Z 274.606,A -85,B 0,C 180,E1 -5437.346,E2 -5437.346} C_VEL
LIN {X 0,Y 509.804,Z 274.608,A -85,B 0,C 180,E1 -5440.386,E2 -5440.386} C_VEL
LIN {X 0,Y 509.799,Z 274.605,A -85,B 0,C 180,E1 -5443.575,E2 -5443.575} C_VEL
LIN {X 0,Y 509.787,Z 274.609,A -85,B 0,C 180,E1 -5446.426,E2 -5446.426} C_VEL
LIN {X 0,Y 509.809,Z 274.606,A -85,B 0,C 180,E1 -5449.616,E2 -5449.616} C_VEL
LIN {X 0,Y 509.779,Z 274.604,A -85,B 0,C 180,E1 -5452.657,E2 -5452.657} C_VEL
LIN {X 0,Y 509.842,Z 274.602,A -85,B 0,C 180,E1 -5455.801,E2 -5455.801} C_VEL
LIN {X 0,Y 509.843,Z 274.6,A -85,B 0,C 180,E1 -5458.721,E2 -5458.721} C_VEL
LIN {X 0,Y 509.877,Z 274.633,A -85,B 0,C 180,E1 -5461.447,E2 -5461.447} C_VEL
LIN {X 0,Y 513.036,Z 288.407,A -85,B 0,C 180,E1 -5463.564,E2 -5463.564} C_VEL
LIN {X 0,Y 512.722,Z 300.987,A -85,B 0,C 180,E1 -5465.288,E2 -5465.288} C_VEL
LIN {X 0,Y 512.033,Z 320.419,A -85,B 0,C 180,E1 -5467.899,E2 -5467.899} C_VEL
LIN {X 0,Y 515.261,Z 337.339,A -85,B 0,C 180,E1 -5468.297,E2 -5468.297} C_VEL
LIN {X 0,Y 514.086,Z 486.401,A -85,B 0,C 180,E1 -5470.459,E2 -5470.459} C_VEL
LIN {X 0,Y 513.717,Z 501.855,A -85,B 0,C 180,E1 -5470.833,E2 -5470.833} C_VEL
LIN {X 0,Y 513.317,Z 517.475,A -85,B 0,C 180,E1 -5471.389,E2 -5471.389} C_VEL
LIN {X 0,Y 512.764,Z 531.329,A -85,B 0,C 180,E1 -5472.039,E2 -5472.039} C_VEL
LIN {X 0,Y 512.223,Z 544.945,A -85,B 0,C 180,E1 -5472.844,E2 -5472.844} C_VEL
LIN {X 0,Y 511.707,Z 557.487,A -85,B 0,C 180,E1 -5473.75,E2 -5473.75} C_VEL
LIN {X 0,Y 511.134,Z 570.229,A -85,B 0,C 180,E1 -5474.857,E2 -5474.857} C_VEL
LIN {X 0,Y 510.613,Z 581.801,A -85,B 0,C 180,E1 -5476.063,E2 -5476.063} C_VEL
LIN {X 0,Y 510.225,Z 591.54,A -85,B 0,C 180,E1 -5477.269,E2 -5477.269} C_VEL
LIN {X 0,Y 509.85,Z 601.257,A -85,B 0,C 180,E1 -5478.698,E2 -5478.698} C_VEL
LIN {X 0,Y 509.565,Z 609.065,A -85,B 0,C 180,E1 -5480.073,E2 -5480.073} C_VEL
LIN {X 0,Y 509.402,Z 616.5,A -85,B 0,C 180,E1 -5481.671,E2 -5481.671} C_VEL
LIN {X 0,Y 509.278,Z 622.397,A -85,B 0,C 180,E1 -5483.265,E2 -5483.265} C_VEL
LIN {X 0,Y 509.262,Z 625.899,A -85,B 0,C 180,E1 -5484.457,E2 -5484.457} C_VEL
LIN {X 0,Y 509.186,Z 629.44,A -85,B 0,C 180,E1 -5486.043,E2 -5486.043} C_VEL
LIN {X 0,Y 509.187,Z 631.77,A -85,B 0,C 180,E1 -5487.627,E2 -5487.627} C_VEL
LIN {X 0,Y 509.071,Z 632.941,A -85,B 0,C 180,E1 -5489.209,E2 -5489.209} C_VEL
LIN {X 0,Y 509.071,Z 632.942,A -85,B 0,C 180,E1 -5490.791,E2 -5490.791} C_VEL
LIN {X 0,Y 509.187,Z 631.772,A -85,B 0,C 180,E1 -5492.373,E2 -5492.373} C_VEL
LIN {X 0,Y 509.186,Z 629.446,A -85,B 0,C 180,E1 -5493.957,E2 -5493.957} C_VEL
LIN {X 0,Y 509.262,Z 625.917,A -85,B 0,C 180,E1 -5495.544,E2 -5495.544} C_VEL
LIN {X 0,Y 509.316,Z 621.091,A -85,B 0,C 180,E1 -5497.134,E2 -5497.134} C_VEL
LIN {X 0,Y 509.443,Z 614.84,A -85,B 0,C 180,E1 -5498.728,E2 -5498.728} C_VEL
LIN {X 0,Y 509.706,Z 606.99,A -85,B 0,C 180,E1 -5500.326,E2 -5500.326} C_VEL
LIN {X 0,Y 509.96,Z 598.493,A -85,B 0,C 180,E1 -5501.75,E2 -5501.75} C_VEL
LIN {X 0,Y 510.357,Z 588.573,A -85,B 0,C 180,E1 -5503.133,E2 -5503.133} C_VEL
LIN {X 0,Y 510.773,Z 578.285,A -85,B 0,C 180,E1 -5504.34,E2 -5504.34} C_VEL
LIN {X 0,Y 511.31,Z 566.83,A -85,B 0,C 180,E1 -5505.47,E2 -5505.47} C_VEL
LIN {X 0,Y 511.87,Z 553.703,A -85,B 0,C 180,E1 -5506.553,E2 -5506.553} C_VEL
LIN {X 0,Y 512.491,Z 540.296,A -85,B 0,C 180,E1 -5507.456,E2 -5507.456} C_VEL
LIN {X 0,Y 513.032,Z 525.487,A -85,B 0,C 180,E1 -5508.262,E2 -5508.262} C_VEL
LIN {X 0,Y 513.544,Z 509.995,A -85,B 0,C 180,E1 -5508.907,E2 -5508.907} C_VEL
LIN {X 0,Y 513.924,Z 494.6,A -85,B 0,C 180,E1 -5509.37,E2 -5509.37} C_VEL
LIN {X 0,Y 514.167,Z 478.244,A -85,B 0,C 180,E1 -5509.681,E2 -5509.681} C_VEL
LIN {X 0,Y 515.305,Z 337.508,A -85,B 0,C 180,E1 -5511.702,E2 -5511.702} C_VEL
LIN {X 0,Y 512.029,Z 320.639,A -85,B 0,C 180,E1 -5512.104,E2 -5512.104} C_VEL
LIN {X 0,Y 512.871,Z 299.687,A -85,B 0,C 180,E1 -5514.921,E2 -5514.921} C_VEL
LIN {X 0,Y 513.101,Z 288.69,A -85,B 0,C 180,E1 -5516.433,E2 -5516.433} C_VEL
LIN {X 0,Y 509.873,Z 274.598,A -85,B 0,C 180,E1 -5518.604,E2 -5518.604} C_VEL
LIN {X 0,Y 509.82,Z 274.604,A -85,B 0,C 180,E1 -5521.59,E2 -5521.59} C_VEL
LIN {X 0,Y 509.834,Z 274.607,A -85,B 0,C 180,E1 -5524.414,E2 -5524.414} C_VEL
LIN {X 0,Y 509.794,Z 274.607,A -85,B 0,C 180,E1 -5527.342,E2 -5527.342} C_VEL
LIN {X 0,Y 509.813,Z 274.606,A -85,B 0,C 180,E1 -5530.384,E2 -5530.384} C_VEL
LIN {X 0,Y 509.804,Z 274.603,A -85,B 0,C 180,E1 -5533.573,E2 -5533.573} C_VEL
LIN {X 0,Y 509.806,Z 274.605,A -85,B 0,C 180,E1 -5536.426,E2 -5536.426} C_VEL
LIN {X 0,Y 509.81,Z 274.605,A -85,B 0,C 180,E1 -5539.305,E2 -5539.305} C_VEL
LIN {X 0,Y 509.811,Z 274.606,A -85,B 0,C 180,E1 -5541.791,E2 -5541.791} C_VEL
LIN {X 0,Y 509.805,Z 274.601,A -85,B 0,C 180,E1 -5544.619,E2 -5544.619} C_VEL
LIN {X 0,Y 509.857,Z 274.597,A -85,B 0,C 180,E1 -5547.48,E2 -5547.48} C_VEL
LIN {X 0,Y 509.855,Z 274.599,A -85,B 0,C 180,E1 -5550.273,E2 -5550.273} C_VEL
LIN {X 0,Y 509.816,Z 274.599,A -85,B 0,C 180,E1 -5552.94,E2 -5552.94} C_VEL
LIN {X 0,Y 509.829,Z 274.606,A -85,B 0,C 180,E1 -5555.571,E2 -5555.571} C_VEL
LIN {X 0,Y 509.817,Z 274.606,A -85,B 0,C 180,E1 -5558.147,E2 -5558.147} C_VEL
LIN {X 0,Y 509.849,Z 274.596,A -85,B 0,C 180,E1 -5560.68,E2 -5560.68} C_VEL
LIN {X 0,Y 509.846,Z 274.6,A -85,B 0,C 180,E1 -5563.172,E2 -5563.172} C_VEL
LIN {X 0,Y 509.851,Z 274.598,A -85,B 0,C 180,E1 -5565.633,E2 -5565.633} C_VEL
LIN {X 0,Y 509.883,Z 274.588,A -85,B 0,C 180,E1 -5568.13,E2 -5568.13} C_VEL
LIN {X 0,Y 509.864,Z 274.597,A -85,B 0,C 180,E1 -5571.278,E2 -5571.278} C_VEL
LIN {X 0,Y 509.911,Z 274.594,A -85,B 0,C 180,E1 -5573.668,E2 -5573.668} C_VEL
LIN {X 0,Y 509.875,Z 274.583,A -85,B 0,C 180,E1 -5576.838,E2 -5576.838} C_VEL
LIN {X 0,Y 509.909,Z 274.584,A -85,B 0,C 180,E1 -5578.419,E2 -5578.419} C_VEL
LIN {X 0,Y 510.018,Z 274.577,A -85,B 0,C 180,E1 -5579.999,E2 -5579.999} C_VEL
LIN {X 0,Y 510.03,Z 274.573,A -85,B 0,C 180,E1 -5582.368,E2 -5582.368} C_VEL
LIN {X 0,Y 509.917,Z 274.584,A -85,B 0,C 180,E1 -5585.535,E2 -5585.535} C_VEL
LIN {X 0,Y 509.859,Z 274.59,A -85,B 0,C 180,E1 -5588.72,E2 -5588.72} C_VEL
LIN {X 0,Y 509.893,Z 274.593,A -85,B 0,C 180,E1 -5591.93,E2 -5591.93} C_VEL
LIN {X 0,Y 509.884,Z 274.593,A -85,B 0,C 180,E1 -5595.24,E2 -5595.24} C_VEL
LIN {X 0,Y 509.822,Z 274.592,A -85,B 0,C 180,E1 -5598.483,E2 -5598.483} C_VEL
LIN {X 0,Y 509.83,Z 274.601,A -85,B 0,C 180,E1 -5601.001,E2 -5601.001} C_VEL
LIN {X 0,Y 509.804,Z 274.604,A -85,B 0,C 180,E1 -5603.563,E2 -5603.563} C_VEL
LIN {X 0,Y 509.803,Z 274.593,A -85,B 0,C 180,E1 -5606.355,E2 -5606.355} C_VEL
LIN {X 0,Y 509.821,Z 274.595,A -85,B 0,C 180,E1 -5608.846,E2 -5608.846} C_VEL
LIN {X 0,Y 509.803,Z 274.605,A -85,B 0,C 180,E1 -5611.589,E2 -5611.589} C_VEL
LIN {X 0,Y 509.818,Z 274.598,A -85,B 0,C 180,E1 -5614.414,E2 -5614.414} C_VEL
LIN {X 0,Y 509.791,Z 274.603,A -85,B 0,C 180,E1 -5617.341,E2 -5617.341} C_VEL
LIN {X 0,Y 509.813,Z 274.601,A -85,B 0,C 180,E1 -5620.382,E2 -5620.382} C_VEL
LIN {X 0,Y 509.782,Z 274.61,A -85,B 0,C 180,E1 -5623.058,E2 -5623.058} C_VEL
LIN {X 0,Y 509.804,Z 274.596,A -85,B 0,C 180,E1 -5625.792,E2 -5625.792} C_VEL
LIN {X 0,Y 509.834,Z 274.601,A -85,B 0,C 180,E1 -5628.573,E2 -5628.573} C_VEL
LIN {X 0,Y 509.832,Z 274.595,A -85,B 0,C 180,E1 -5631.786,E2 -5631.786} C_VEL
LIN {X 0,Y 509.805,Z 274.599,A -85,B 0,C 180,E1 -5633.681,E2 -5633.681} C_VEL
LIN {X 0,Y 509.136,Z 274.684,A -85,B 0,C 180,E1 -5634.341,E2 -5634.341} C_VEL
LIN {X 0,Y 506.326,Z 275.041,A -85,B 0,C 180,E1 -5635.412,E2 -5635.412} C_VEL
LIN {X 0,Y 503.941,Z 275.342,A -85,B 0,C 180,E1 -5636.276,E2 -5636.276} C_VEL
LIN {X 0,Y 502.893,Z 275.471,A -85,B 0,C 180,E1 -5636.942,E2 -5636.942} C_VEL
LIN {X 0,Y 502.793,Z 275.48,A -85,B 0,C 180,E1 -5637.168,E2 -5637.168} C_VEL
LIN {X 0,Y 502.796,Z 275.47,A -85,B 0,C 180,E1 -5640.064,E2 -5640.064} C_VEL
LIN {X 0,Y 502.81,Z 275.477,A -85,B 0,C 180,E1 -5642.532,E2 -5642.532} C_VEL
LIN {X 0,Y 502.768,Z 275.48,A -85,B 0,C 180,E1 -5645.308,E2 -5645.308} C_VEL
LIN {X 0,Y 502.761,Z 275.48,A -85,B 0,C 180,E1 -5647.826,E2 -5647.826} C_VEL
LIN {X 0,Y 502.806,Z 275.475,A -85,B 0,C 180,E1 -5650.4,E2 -5650.4} C_VEL
LIN {X 0,Y 502.81,Z 275.477,A -85,B 0,C 180,E1 -5652.931,E2 -5652.931} C_VEL
LIN {X 0,Y 502.825,Z 275.472,A -85,B 0,C 180,E1 -5655.429,E2 -5655.429} C_VEL
LIN {X 0,Y 502.88,Z 275.471,A -85,B 0,C 180,E1 -5658.717,E2 -5658.717} C_VEL
LIN {X 0,Y 502.881,Z 275.465,A -85,B 0,C 180,E1 -5661.966,E2 -5661.966} C_VEL
LIN {X 0,Y 502.914,Z 275.466,A -85,B 0,C 180,E1 -5664.386,E2 -5664.386} C_VEL
LIN {X 0,Y 503.003,Z 275.452,A -85,B 0,C 180,E1 -5667.597,E2 -5667.597} C_VEL
LIN {X 0,Y 503.004,Z 275.456,A -85,B 0,C 180,E1 -5670,E2 -5670} C_VEL
LIN {X 0,Y 503.004,Z 275.46,A -85,B 0,C 180,E1 -5672.402,E2 -5672.402} C_VEL
LIN {X 0,Y 502.838,Z 275.515,A -85,B 0,C 180,E1 -5674.459,E2 -5674.459} C_VEL
LIN {X 0,Y 505.234,Z 286.572,A -85,B 0,C 180,E1 -5676.389,E2 -5676.389} C_VEL
LIN {X 0,Y 505.417,Z 290.233,A -85,B 0,C 180,E1 -5676.988,E2 -5676.988} C_VEL
LIN {X 0,Y 505.26,Z 294.372,A -85,B 0,C 180,E1 -5677.643,E2 -5677.643} C_VEL
LIN {X 0,Y 508.781,Z 310.974,A -85,B 0,C 180,E1 -5678.064,E2 -5678.064} C_VEL
LIN {X 0,Y 507.48,Z 459.45,A -85,B 0,C 180,E1 -5680.252,E2 -5680.252} C_VEL
LIN {X 0,Y 507.141,Z 474.579,A -85,B 0,C 180,E1 -5680.63,E2 -5680.63} C_VEL
LIN {X 0,Y 506.657,Z 490.187,A -85,B 0,C 180,E1 -5681.197,E2 -5681.197} C_VEL
LIN {X 0,Y 506.159,Z 504.97,A -85,B 0,C 180,E1 -5681.919,E2 -5681.919} C_VEL
LIN {X 0,Y 505.578,Z 518.458,A -85,B 0,C 180,E1 -5682.748,E2 -5682.748} C_VEL
LIN {X 0,Y 504.912,Z 532.213,A -85,B 0,C 180,E1 -5683.79,E2 -5683.79} C_VEL
LIN {X 0,Y 504.337,Z 544.652,A -85,B 0,C 180,E1 -5684.939,E2 -5684.939} C_VEL
LIN {X 0,Y 503.742,Z 556.047,A -85,B 0,C 180,E1 -5686.202,E2 -5686.202} C_VEL
LIN {X 0,Y 503.283,Z 565.653,A -85,B 0,C 180,E1 -5687.471,E2 -5687.471} C_VEL
LIN {X 0,Y 502.86,Z 575.086,A -85,B 0,C 180,E1 -5688.961,E2 -5688.961} C_VEL
LIN {X 0,Y 502.566,Z 582.91,A -85,B 0,C 180,E1 -5690.462,E2 -5690.462} C_VEL
LIN {X 0,Y 502.367,Z 588.51,A -85,B 0,C 180,E1 -5691.76,E2 -5691.76} C_VEL
LIN {X 0,Y 502.209,Z 594.565,A -85,B 0,C 180,E1 -5693.504,E2 -5693.504} C_VEL
LIN {X 0,Y 502.155,Z 598.12,A -85,B 0,C 180,E1 -5694.825,E2 -5694.825} C_VEL
LIN {X 0,Y 502.002,Z 601.575,A -85,B 0,C 180,E1 -5696.614,E2 -5696.614} C_VEL
LIN {X 0,Y 501.975,Z 603.59,A -85,B 0,C 180,E1 -5698.425,E2 -5698.425} C_VEL
LIN {X 0,Y 501.982,Z 604.143,A -85,B 0,C 180,E1 -5699.774,E2 -5699.774} C_VEL
LIN {X 0,Y 501.979,Z 603.783,A -85,B 0,C 180,E1 -5701.351,E2 -5701.351} C_VEL
LIN {X 0,Y 501.993,Z 602.125,A -85,B 0,C 180,E1 -5703.092,E2 -5703.092} C_VEL
LIN {X 0,Y 502.048,Z 600.144,A -85,B 0,C 180,E1 -5704.322,E2 -5704.322} C_VEL
LIN {X 0,Y 502.182,Z 596.271,A -85,B 0,C 180,E1 -5705.999,E2 -5705.999} C_VEL
LIN {X 0,Y 502.277,Z 591.57,A -85,B 0,C 180,E1 -5707.516,E2 -5707.516} C_VEL
LIN {X 0,Y 502.47,Z 585.765,A -85,B 0,C 180,E1 -5709.005,E2 -5709.005} C_VEL
LIN {X 0,Y 502.736,Z 578.51,A -85,B 0,C 180,E1 -5710.516,E2 -5710.516} C_VEL
LIN {X 0,Y 503.039,Z 570.858,A -85,B 0,C 180,E1 -5711.844,E2 -5711.844} C_VEL
LIN {X 0,Y 503.517,Z 560.652,A -85,B 0,C 180,E1 -5713.316,E2 -5713.316} C_VEL
LIN {X 0,Y 504.063,Z 549.227,A -85,B 0,C 180,E1 -5714.68,E2 -5714.68} C_VEL
LIN {X 0,Y 504.7,Z 537.153,A -85,B 0,C 180,E1 -5715.876,E2 -5715.876} C_VEL
LIN {X 0,Y 505.34,Z 523.97,A -85,B 0,C 180,E1 -5716.954,E2 -5716.954} C_VEL
LIN {X 0,Y 505.91,Z 510.606,A -85,B 0,C 180,E1 -5717.852,E2 -5717.852} C_VEL
LIN {X 0,Y 506.466,Z 496.595,A -85,B 0,C 180,E1 -5718.606,E2 -5718.606} C_VEL
LIN {X 0,Y 506.951,Z 481.262,A -85,B 0,C 180,E1 -5719.24,E2 -5719.24} C_VEL
LIN {X 0,Y 507.364,Z 466.381,A -85,B 0,C 180,E1 -5719.684,E2 -5719.684} C_VEL
LIN {X 0,Y 507.573,Z 451.77,A -85,B 0,C 180,E1 -5719.97,E2 -5719.97} C_VEL
LIN {X 0,Y 508.7,Z 309.885,A -85,B 0,C 180,E1 -5722.05,E2 -5722.05} C_VEL
LIN {X 0,Y 505.265,Z 294.688,A -85,B 0,C 180,E1 -5722.45,E2 -5722.45} C_VEL
LIN {X 0,Y 505.379,Z 287.301,A -85,B 0,C 180,E1 -5723.632,E2 -5723.632} C_VEL
LIN {X 0,Y 502.814,Z 275.48,A -85,B 0,C 180,E1 -5725.72,E2 -5725.72} C_VEL
LIN {X 0,Y 502.782,Z 275.482,A -85,B 0,C 180,E1 -5728.858,E2 -5728.858} C_VEL
LIN {X 0,Y 502.828,Z 275.478,A -85,B 0,C 180,E1 -5731.705,E2 -5731.705} C_VEL
LIN {X 0,Y 502.825,Z 275.474,A -85,B 0,C 180,E1 -5734.326,E2 -5734.326} C_VEL
LIN {X 0,Y 502.782,Z 275.484,A -85,B 0,C 180,E1 -5737.3,E2 -5737.3} C_VEL
LIN {X 0,Y 502.81,Z 275.475,A -85,B 0,C 180,E1 -5740.401,E2 -5740.401} C_VEL
LIN {X 0,Y 502.821,Z 275.479,A -85,B 0,C 180,E1 -5742.933,E2 -5742.933} C_VEL
LIN {X 0,Y 502.83,Z 275.477,A -85,B 0,C 180,E1 -5745.43,E2 -5745.43} C_VEL
LIN {X 0,Y 502.862,Z 275.471,A -85,B 0,C 180,E1 -5748.718,E2 -5748.718} C_VEL
LIN {X 0,Y 502.886,Z 275.464,A -85,B 0,C 180,E1 -5751.968,E2 -5751.968} C_VEL
LIN {X 0,Y 502.919,Z 275.46,A -85,B 0,C 180,E1 -5754.388,E2 -5754.388} C_VEL
LIN {X 0,Y 503.008,Z 275.451,A -85,B 0,C 180,E1 -5757.599,E2 -5757.599} C_VEL
LIN {X 0,Y 503.01,Z 275.449,A -85,B 0,C 180,E1 -5760.001,E2 -5760.001} C_VEL
LIN {X 0,Y 503.009,Z 275.449,A -85,B 0,C 180,E1 -5762.404,E2 -5762.404} C_VEL
LIN {X 0,Y 502.911,Z 275.461,A -85,B 0,C 180,E1 -5765.615,E2 -5765.615} C_VEL
LIN {X 0,Y 502.867,Z 275.465,A -85,B 0,C 180,E1 -5768.035,E2 -5768.035} C_VEL
LIN {X 0,Y 502.865,Z 275.468,A -85,B 0,C 180,E1 -5771.285,E2 -5771.285} C_VEL
LIN {X 0,Y 502.832,Z 275.476,A -85,B 0,C 180,E1 -5774.572,E2 -5774.572} C_VEL
LIN {X 0,Y 502.812,Z 275.473,A -85,B 0,C 180,E1 -5777.91,E2 -5777.91} C_VEL
LIN {X 0,Y 502.82,Z 275.478,A -85,B 0,C 180,E1 -5780.537,E2 -5780.537} C_VEL
LIN {X 0,Y 502.777,Z 275.478,A -85,B 0,C 180,E1 -5783.042,E2 -5783.042} C_VEL
LIN {X 0,Y 502.76,Z 275.479,A -85,B 0,C 180,E1 -5785.681,E2 -5785.681} C_VEL
LIN {X 0,Y 502.785,Z 275.482,A -85,B 0,C 180,E1 -5788.377,E2 -5788.377} C_VEL
LIN {X 0,Y 502.777,Z 275.476,A -85,B 0,C 180,E1 -5791.145,E2 -5791.145} C_VEL
LIN {X 0,Y 502.777,Z 275.481,A -85,B 0,C 180,E1 -5793.997,E2 -5793.997} C_VEL
LIN {X 0,Y 502.724,Z 275.483,A -85,B 0,C 180,E1 -5797.172,E2 -5797.172} C_VEL
LIN {X 0,Y 502.761,Z 275.484,A -85,B 0,C 180,E1 -5800.019,E2 -5800.019} C_VEL
LIN {X 0,Y 502.74,Z 275.483,A -85,B 0,C 180,E1 -5803.236,E2 -5803.236} C_VEL
LIN {X 0,Y 502.762,Z 275.483,A -85,B 0,C 180,E1 -5805.66,E2 -5805.66} C_VEL
LIN {X 0,Y 502.759,Z 275.481,A -85,B 0,C 180,E1 -5809.014,E2 -5809.014} C_VEL
LIN {X 0,Y 502.757,Z 275.486,A -85,B 0,C 180,E1 -5812.044,E2 -5812.044} C_VEL
LIN {X 0,Y 502.785,Z 275.478,A -85,B 0,C 180,E1 -5815.034,E2 -5815.034} C_VEL
LIN {X 0,Y 502.78,Z 275.485,A -85,B 0,C 180,E1 -5817.916,E2 -5817.916} C_VEL
LIN {X 0,Y 502.856,Z 275.591,A -85,B 0,C 180,E1 -5821.174,E2 -5821.174} C_VEL
LIN {X 0,Y 506.2,Z 290.071,A -85,B 0,C 180,E1 -5823.441,E2 -5823.441} C_VEL
LIN {X 0,Y 505.883,Z 302.39,A -85,B 0,C 180,E1 -5825.155,E2 -5825.155} C_VEL
LIN {X 0,Y 505.183,Z 320.17,A -85,B 0,C 180,E1 -5827.58,E2 -5827.58} C_VEL
LIN {X 0,Y 508.682,Z 339.241,A -85,B 0,C 180,E1 -5828.034,E2 -5828.034} C_VEL
LIN {X 0,Y 507.38,Z 486.779,A -85,B 0,C 180,E1 -5830.205,E2 -5830.205} C_VEL
LIN {X 0,Y 506.975,Z 502.375,A -85,B 0,C 180,E1 -5830.595,E2 -5830.595} C_VEL
LIN {X 0,Y 506.554,Z 517.522,A -85,B 0,C 180,E1 -5831.146,E2 -5831.146} C_VEL
LIN {X 0,Y 505.975,Z 531.034,A -85,B 0,C 180,E1 -5831.789,E2 -5831.789} C_VEL
LIN {X 0,Y 505.388,Z 544.666,A -85,B 0,C 180,E1 -5832.604,E2 -5832.604} C_VEL
LIN {X 0,Y 504.808,Z 557.221,A -85,B 0,C 180,E1 -5833.522,E2 -5833.522} C_VEL
LIN {X 0,Y 504.208,Z 569.974,A -85,B 0,C 180,E1 -5834.644,E2 -5834.644} C_VEL
LIN {X 0,Y 503.665,Z 581.555,A -85,B 0,C 180,E1 -5835.867,E2 -5835.867} C_VEL
LIN {X 0,Y 503.208,Z 591.301,A -85,B 0,C 180,E1 -5837.088,E2 -5837.088} C_VEL
LIN {X 0,Y 502.808,Z 601.063,A -85,B 0,C 180,E1 -5838.544,E2 -5838.544} C_VEL
LIN {X 0,Y 502.527,Z 608.84,A -85,B 0,C 180,E1 -5839.933,E2 -5839.933} C_VEL
LIN {X 0,Y 502.325,Z 616.28,A -85,B 0,C 180,E1 -5841.553,E2 -5841.553} C_VEL
LIN {X 0,Y 502.198,Z 622.181,A -85,B 0,C 180,E1 -5843.169,E2 -5843.169} C_VEL
LIN {X 0,Y 502.172,Z 625.688,A -85,B 0,C 180,E1 -5844.378,E2 -5844.378} C_VEL
LIN {X 0,Y 502.082,Z 629.231,A -85,B 0,C 180,E1 -5845.987,E2 -5845.987} C_VEL
LIN {X 0,Y 502.088,Z 631.565,A -85,B 0,C 180,E1 -5847.594,E2 -5847.594} C_VEL
LIN {X 0,Y 501.988,Z 632.738,A -85,B 0,C 180,E1 -5849.198,E2 -5849.198} C_VEL
LIN {X 0,Y 501.988,Z 632.74,A -85,B 0,C 180,E1 -5850.802,E2 -5850.802} C_VEL
LIN {X 0,Y 502.088,Z 631.57,A -85,B 0,C 180,E1 -5852.407,E2 -5852.407} C_VEL
LIN {X 0,Y 502.082,Z 629.242,A -85,B 0,C 180,E1 -5854.014,E2 -5854.014} C_VEL
LIN {X 0,Y 502.172,Z 625.712,A -85,B 0,C 180,E1 -5855.622,E2 -5855.622} C_VEL
LIN {X 0,Y 502.241,Z 620.884,A -85,B 0,C 180,E1 -5857.235,E2 -5857.235} C_VEL
LIN {X 0,Y 502.36,Z 614.629,A -85,B 0,C 180,E1 -5858.853,E2 -5858.853} C_VEL
LIN {X 0,Y 502.652,Z 606.776,A -85,B 0,C 180,E1 -5860.473,E2 -5860.473} C_VEL
LIN {X 0,Y 502.911,Z 598.826,A -85,B 0,C 180,E1 -5861.832,E2 -5861.832} C_VEL
LIN {X 0,Y 503.379,Z 588.349,A -85,B 0,C 180,E1 -5863.319,E2 -5863.319} C_VEL
LIN {X 0,Y 503.809,Z 578.057,A -85,B 0,C 180,E1 -5864.542,E2 -5864.542} C_VEL
LIN {X 0,Y 504.451,Z 565.805,A -85,B 0,C 180,E1 -5865.762,E2 -5865.762} C_VEL
LIN {X 0,Y 505.053,Z 552.098,A -85,B 0,C 180,E1 -5866.887,E2 -5866.887} C_VEL
LIN {X 0,Y 505.752,Z 538.38,A -85,B 0,C 180,E1 -5867.801,E2 -5867.801} C_VEL
LIN {X 0,Y 506.282,Z 524.149,A -85,B 0,C 180,E1 -5868.567,E2 -5868.567} C_VEL
LIN {X 0,Y 506.838,Z 509.168,A -85,B 0,C 180,E1 -5869.186,E2 -5869.186} C_VEL
LIN {X 0,Y 507.211,Z 494.264,A -85,B 0,C 180,E1 -5869.636,E2 -5869.636} C_VEL
LIN {X 0,Y 507.471,Z 477.824,A -85,B 0,C 180,E1 -5869.952,E2 -5869.952} C_VEL
LIN {X 0,Y 508.713,Z 338.678,A -85,B 0,C 180,E1 -5871.977,E2 -5871.977} C_VEL
LIN {X 0,Y 505.199,Z 320.447,A -85,B 0,C 180,E1 -5872.419,E2 -5872.419} C_VEL
LIN {X 0,Y 506.069,Z 299.973,A -85,B 0,C 180,E1 -5875.213,E2 -5875.213} C_VEL
LIN {X 0,Y 506.282,Z 290.332,A -85,B 0,C 180,E1 -5876.559,E2 -5876.559} C_VEL
LIN {X 0,Y 502.847,Z 275.476,A -85,B 0,C 180,E1 -5878.885,E2 -5878.885} C_VEL
LIN {X 0,Y 502.783,Z 275.484,A -85,B 0,C 180,E1 -5882.084,E2 -5882.084} C_VEL
LIN {X 0,Y 502.79,Z 275.48,A -85,B 0,C 180,E1 -5884.966,E2 -5884.966} C_VEL
LIN {X 0,Y 502.764,Z 275.485,A -85,B 0,C 180,E1 -5888.481,E2 -5888.481} C_VEL
LIN {X 0,Y 502.763,Z 275.479,A -85,B 0,C 180,E1 -5891.071,E2 -5891.071} C_VEL
LIN {X 0,Y 502.784,Z 275.48,A -85,B 0,C 180,E1 -5894.529,E2 -5894.529} C_VEL
LIN {X 0,Y 502.765,Z 275.485,A -85,B 0,C 180,E1 -5897.857,E2 -5897.857} C_VEL
LIN {X 0,Y 502.78,Z 275.475,A -85,B 0,C 180,E1 -5901.021,E2 -5901.021} C_VEL
LIN {X 0,Y 502.748,Z 275.484,A -85,B 0,C 180,E1 -5904.172,E2 -5904.172} C_VEL
LIN {X 0,Y 502.801,Z 275.473,A -85,B 0,C 180,E1 -5906.998,E2 -5906.998} C_VEL
LIN {X 0,Y 502.811,Z 275.48,A -85,B 0,C 180,E1 -5910.064,E2 -5910.064} C_VEL
LIN {X 0,Y 502.778,Z 275.479,A -85,B 0,C 180,E1 -5913.428,E2 -5913.428} C_VEL
LIN {X 0,Y 502.762,Z 275.484,A -85,B 0,C 180,E1 -5916.084,E2 -5916.084} C_VEL
LIN {X 0,Y 502.779,Z 275.479,A -85,B 0,C 180,E1 -5918.688,E2 -5918.688} C_VEL
LIN {X 0,Y 502.805,Z 275.475,A -85,B 0,C 180,E1 -5921.246,E2 -5921.246} C_VEL
LIN {X 0,Y 502.832,Z 275.469,A -85,B 0,C 180,E1 -5924.663,E2 -5924.663} C_VEL
LIN {X 0,Y 502.864,Z 275.463,A -85,B 0,C 180,E1 -5928.042,E2 -5928.042} C_VEL
LIN {X 0,Y 502.827,Z 275.472,A -85,B 0,C 180,E1 -5931.155,E2 -5931.155} C_VEL
LIN {X 0,Y 502.861,Z 275.473,A -85,B 0,C 180,E1 -5933.579,E2 -5933.579} C_VEL
LIN {X 0,Y 502.82,Z 275.461,A -85,B 0,C 180,E1 -5936.794,E2 -5936.794} C_VEL
LIN {X 0,Y 502.879,Z 275.46,A -85,B 0,C 180,E1 -5938.397,E2 -5938.397} C_VEL
LIN {X 0,Y 502.987,Z 275.453,A -85,B 0,C 180,E1 -5939.999,E2 -5939.999} C_VEL
LIN {X 0,Y 503,Z 275.449,A -85,B 0,C 180,E1 -5942.401,E2 -5942.401} C_VEL
LIN {X 0,Y 502.871,Z 275.459,A -85,B 0,C 180,E1 -5945.613,E2 -5945.613} C_VEL
LIN {X 0,Y 502.823,Z 275.467,A -85,B 0,C 180,E1 -5948.843,E2 -5948.843} C_VEL
LIN {X 0,Y 502.832,Z 275.471,A -85,B 0,C 180,E1 -5952.1,E2 -5952.1} C_VEL
LIN {X 0,Y 502.835,Z 275.467,A -85,B 0,C 180,E1 -5955.398,E2 -5955.398} C_VEL
LIN {X 0,Y 502.795,Z 275.469,A -85,B 0,C 180,E1 -5958.751,E2 -5958.751} C_VEL
LIN {X 0,Y 502.766,Z 275.486,A -85,B 0,C 180,E1 -5961.31,E2 -5961.31} C_VEL
LIN {X 0,Y 502.753,Z 275.479,A -85,B 0,C 180,E1 -5963.914,E2 -5963.914} C_VEL
LIN {X 0,Y 502.77,Z 275.469,A -85,B 0,C 180,E1 -5966.569,E2 -5966.569} C_VEL
LIN {X 0,Y 502.795,Z 275.474,A -85,B 0,C 180,E1 -5969.933,E2 -5969.933} C_VEL
LIN {X 0,Y 502.787,Z 275.483,A -85,B 0,C 180,E1 -5973.032,E2 -5973.032} C_VEL
LIN {X 0,Y 502.75,Z 275.471,A -85,B 0,C 180,E1 -5975.951,E2 -5975.951} C_VEL
LIN {X 0,Y 502.78,Z 275.478,A -85,B 0,C 180,E1 -5978.975,E2 -5978.975} C_VEL
LIN {X 0,Y 502.754,Z 275.48,A -85,B 0,C 180,E1 -5982.194,E2 -5982.194} C_VEL
LIN {X 0,Y 502.768,Z 275.475,A -85,B 0,C 180,E1 -5985.469,E2 -5985.469} C_VEL
LIN {X 0,Y 502.778,Z 275.477,A -85,B 0,C 180,E1 -5987.859,E2 -5987.859} C_VEL
LIN {X 0,Y 502.783,Z 275.482,A -85,B 0,C 180,E1 -5991.023,E2 -5991.023} C_VEL
LIN {X 0,Y 502.758,Z 275.476,A -85,B 0,C 180,E1 -5994.168,E2 -5994.168} C_VEL
LIN {X 0,Y 502.793,Z 275.48,A -85,B 0,C 180,E1 -5997.168,E2 -5997.168} C_VEL
LIN {X 0,Y 502.088,Z 275.563,A -85,B 0,C 180,E1 -5997.836,E2 -5997.836} C_VEL
LIN {X 0,Y 499.224,Z 275.921,A -85,B 0,C 180,E1 -5998.922,E2 -5998.922} C_VEL
LIN {X 0,Y 496.831,Z 276.215,A -85,B 0,C 180,E1 -5999.797,E2 -5999.797} C_VEL
LIN {X 0,Y 495.812,Z 276.343,A -85,B 0,C 180,E1 -6000.473,E2 -6000.473} C_VEL
LIN {X 0,Y 495.732,Z 276.353,A -85,B 0,C 180,E1 -6000.701,E2 -6000.701} C_VEL
LIN {X 0,Y 495.805,Z 276.348,A -85,B 0,C 180,E1 -6003.25,E2 -6003.25} C_VEL
LIN {X 0,Y 495.723,Z 276.36,A -85,B 0,C 180,E1 -6006.612,E2 -6006.612} C_VEL
LIN {X 0,Y 495.76,Z 276.351,A -85,B 0,C 180,E1 -6009.323,E2 -6009.323} C_VEL
LIN {X 0,Y 495.774,Z 276.351,A -85,B 0,C 180,E1 -6011.828,E2 -6011.828} C_VEL
LIN {X 0,Y 495.805,Z 276.35,A -85,B 0,C 180,E1 -6014.548,E2 -6014.548} C_VEL
LIN {X 0,Y 495.858,Z 276.341,A -85,B 0,C 180,E1 -6017.938,E2 -6017.938} C_VEL
LIN {X 0,Y 495.823,Z 276.347,A -85,B 0,C 180,E1 -6021.03,E2 -6021.03} C_VEL
LIN {X 0,Y 495.841,Z 276.343,A -85,B 0,C 180,E1 -6023.489,E2 -6023.489} C_VEL
LIN {X 0,Y 495.826,Z 276.353,A -85,B 0,C 180,E1 -6026.749,E2 -6026.749} C_VEL
LIN {X 0,Y 495.987,Z 276.33,A -85,B 0,C 180,E1 -6029.188,E2 -6029.188} C_VEL
LIN {X 0,Y 495.85,Z 276.347,A -85,B 0,C 180,E1 -6031.624,E2 -6031.624} C_VEL
LIN {X 0,Y 495.826,Z 276.351,A -85,B 0,C 180,E1 -6033.25,E2 -6033.25} C_VEL
LIN {X 0,Y 495.781,Z 276.56,A -85,B 0,C 180,E1 -6034.217,E2 -6034.217} C_VEL
LIN {X 0,Y 498.155,Z 286.992,A -85,B 0,C 180,E1 -6036.073,E2 -6036.073} C_VEL
LIN {X 0,Y 498.592,Z 290.555,A -85,B 0,C 180,E1 -6036.678,E2 -6036.678} C_VEL
LIN {X 0,Y 498.446,Z 294.527,A -85,B 0,C 180,E1 -6037.315,E2 -6037.315} C_VEL
LIN {X 0,Y 502.189,Z 311.395,A -85,B 0,C 180,E1 -6037.766,E2 -6037.766} C_VEL
LIN {X 0,Y 500.819,Z 459.398,A -85,B 0,C 180,E1 -6039.976,E2 -6039.976} C_VEL
LIN {X 0,Y 500.442,Z 475.012,A -85,B 0,C 180,E1 -6040.371,E2 -6040.371} C_VEL
LIN {X 0,Y 499.939,Z 490.407,A -85,B 0,C 180,E1 -6040.939,E2 -6040.939} C_VEL
LIN {X 0,Y 499.396,Z 505.194,A -85,B 0,C 180,E1 -6041.671,E2 -6041.671} C_VEL
LIN {X 0,Y 498.784,Z 518.69,A -85,B 0,C 180,E1 -6042.511,E2 -6042.511} C_VEL
LIN {X 0,Y 498.149,Z 531.681,A -85,B 0,C 180,E1 -6043.503,E2 -6043.503} C_VEL
LIN {X 0,Y 497.458,Z 543.868,A -85,B 0,C 180,E1 -6044.627,E2 -6044.627} C_VEL
LIN {X 0,Y 496.884,Z 555.32,A -85,B 0,C 180,E1 -6045.896,E2 -6045.896} C_VEL
LIN {X 0,Y 496.3,Z 565.89,A -85,B 0,C 180,E1 -6047.299,E2 -6047.299} C_VEL
LIN {X 0,Y 495.855,Z 575.388,A -85,B 0,C 180,E1 -6048.823,E2 -6048.823} C_VEL
LIN {X 0,Y 495.538,Z 582.706,A -85,B 0,C 180,E1 -6050.243,E2 -6050.243} C_VEL
LIN {X 0,Y 495.307,Z 588.724,A -85,B 0,C 180,E1 -6051.648,E2 -6051.648} C_VEL
LIN {X 0,Y 495.129,Z 594.778,A -85,B 0,C 180,E1 -6053.417,E2 -6053.417} C_VEL
LIN {X 0,Y 495.073,Z 598.208,A -85,B 0,C 180,E1 -6054.702,E2 -6054.702} C_VEL
LIN {X 0,Y 494.912,Z 601.744,A -85,B 0,C 180,E1 -6056.544,E2 -6056.544} C_VEL
LIN {X 0,Y 494.897,Z 603.734,A -85,B 0,C 180,E1 -6058.307,E2 -6058.307} C_VEL
LIN {X 0,Y 494.899,Z 604.385,A -85,B 0,C 180,E1 -6059.979,E2 -6059.979} C_VEL
LIN {X 0,Y 494.889,Z 603.797,A -85,B 0,C 180,E1 -6061.697,E2 -6061.697} C_VEL
LIN {X 0,Y 494.901,Z 602.39,A -85,B 0,C 180,E1 -6063.091,E2 -6063.091} C_VEL
LIN {X 0,Y 494.98,Z 599.933,A -85,B 0,C 180,E1 -6064.606,E2 -6064.606} C_VEL
LIN {X 0,Y 495.103,Z 596.704,A -85,B 0,C 180,E1 -6065.994,E2 -6065.994} C_VEL
LIN {X 0,Y 495.228,Z 591.83,A -85,B 0,C 180,E1 -6067.605,E2 -6067.605} C_VEL
LIN {X 0,Y 495.437,Z 585.869,A -85,B 0,C 180,E1 -6069.155,E2 -6069.155} C_VEL
LIN {X 0,Y 495.742,Z 578.517,A -85,B 0,C 180,E1 -6070.701,E2 -6070.701} C_VEL
LIN {X 0,Y 496.055,Z 570.992,A -85,B 0,C 180,E1 -6072.021,E2 -6072.021} C_VEL
LIN {X 0,Y 496.501,Z 561.952,A -85,B 0,C 180,E1 -6073.354,E2 -6073.354} C_VEL
LIN {X 0,Y 497.054,Z 551.075,A -85,B 0,C 180,E1 -6074.701,E2 -6074.701} C_VEL
LIN {X 0,Y 497.726,Z 539.269,A -85,B 0,C 180,E1 -6075.918,E2 -6075.918} C_VEL
LIN {X 0,Y 498.39,Z 526.329,A -85,B 0,C 180,E1 -6077.026,E2 -6077.026} C_VEL
LIN {X 0,Y 498.982,Z 513.785,A -85,B 0,C 180,E1 -6077.911,E2 -6077.911} C_VEL
LIN {X 0,Y 499.634,Z 499.585,A -85,B 0,C 180,E1 -6078.721,E2 -6078.721} C_VEL
LIN {X 0,Y 500.143,Z 485.338,A -85,B 0,C 180,E1 -6079.357,E2 -6079.357} C_VEL
LIN {X 0,Y 500.601,Z 470.364,A -85,B 0,C 180,E1 -6079.852,E2 -6079.852} C_VEL
LIN {X 0,Y 500.882,Z 454.83,A -85,B 0,C 180,E1 -6080.194,E2 -6080.194} C_VEL
LIN {X 0,Y 502.226,Z 311.381,A -85,B 0,C 180,E1 -6082.33,E2 -6082.33} C_VEL
LIN {X 0,Y 498.483,Z 294.851,A -85,B 0,C 180,E1 -6082.781,E2 -6082.781} C_VEL
LIN {X 0,Y 498.572,Z 289.209,A -85,B 0,C 180,E1 -6083.7,E2 -6083.7} C_VEL
LIN {X 0,Y 495.762,Z 276.358,A -85,B 0,C 180,E1 -6086.011,E2 -6086.011} C_VEL
LIN {X 0,Y 495.74,Z 276.363,A -85,B 0,C 180,E1 -6089.314,E2 -6089.314} C_VEL
LIN {X 0,Y 495.766,Z 276.355,A -85,B 0,C 180,E1 -6092.11,E2 -6092.11} C_VEL
LIN {X 0,Y 495.772,Z 276.354,A -85,B 0,C 180,E1 -6094.834,E2 -6094.834} C_VEL
LIN {X 0,Y 495.734,Z 276.36,A -85,B 0,C 180,E1 -6097.496,E2 -6097.496} C_VEL
LIN {X 0,Y 495.762,Z 276.353,A -85,B 0,C 180,E1 -6100.111,E2 -6100.111} C_VEL
LIN {X 0,Y 495.772,Z 276.354,A -85,B 0,C 180,E1 -6102.683,E2 -6102.683} C_VEL
LIN {X 0,Y 495.775,Z 276.357,A -85,B 0,C 180,E1 -6105.218,E2 -6105.218} C_VEL
LIN {X 0,Y 495.837,Z 276.345,A -85,B 0,C 180,E1 -6108.556,E2 -6108.556} C_VEL
LIN {X 0,Y 495.858,Z 276.34,A -85,B 0,C 180,E1 -6111.853,E2 -6111.853} C_VEL
LIN {X 0,Y 495.875,Z 276.337,A -85,B 0,C 180,E1 -6114.308,E2 -6114.308} C_VEL
LIN {X 0,Y 495.977,Z 276.327,A -85,B 0,C 180,E1 -6117.565,E2 -6117.565} C_VEL
LIN {X 0,Y 495.981,Z 276.324,A -85,B 0,C 180,E1 -6120.001,E2 -6120.001} C_VEL
LIN {X 0,Y 495.978,Z 276.326,A -85,B 0,C 180,E1 -6122.438,E2 -6122.438} C_VEL
LIN {X 0,Y 495.868,Z 276.339,A -85,B 0,C 180,E1 -6125.695,E2 -6125.695} C_VEL
LIN {X 0,Y 495.824,Z 276.343,A -85,B 0,C 180,E1 -6128.15,E2 -6128.15} C_VEL
LIN {X 0,Y 495.84,Z 276.342,A -85,B 0,C 180,E1 -6131.447,E2 -6131.447} C_VEL
LIN {X 0,Y 495.778,Z 276.356,A -85,B 0,C 180,E1 -6134.784,E2 -6134.784} C_VEL
LIN {X 0,Y 495.753,Z 276.352,A -85,B 0,C 180,E1 -6137.321,E2 -6137.321} C_VEL
LIN {X 0,Y 495.761,Z 276.352,A -85,B 0,C 180,E1 -6139.892,E2 -6139.892} C_VEL
LIN {X 0,Y 495.749,Z 276.356,A -85,B 0,C 180,E1 -6142.861,E2 -6142.861} C_VEL
LIN {X 0,Y 495.703,Z 276.362,A -85,B 0,C 180,E1 -6146.074,E2 -6146.074} C_VEL
LIN {X 0,Y 495.733,Z 276.357,A -85,B 0,C 180,E1 -6148.818,E2 -6148.818} C_VEL
LIN {X 0,Y 495.741,Z 276.354,A -85,B 0,C 180,E1 -6151.725,E2 -6151.725} C_VEL
LIN {X 0,Y 495.747,Z 276.357,A -85,B 0,C 180,E1 -6154.693,E2 -6154.693} C_VEL
LIN {X 0,Y 495.692,Z 276.36,A -85,B 0,C 180,E1 -6157.566,E2 -6157.566} C_VEL
LIN {X 0,Y 495.734,Z 276.36,A -85,B 0,C 180,E1 -6160.046,E2 -6160.046} C_VEL
LIN {X 0,Y 495.689,Z 276.362,A -85,B 0,C 180,E1 -6162.888,E2 -6162.888} C_VEL
LIN {X 0,Y 495.708,Z 276.364,A -85,B 0,C 180,E1 -6165.998,E2 -6165.998} C_VEL
LIN {X 0,Y 495.722,Z 276.358,A -85,B 0,C 180,E1 -6169.297,E2 -6169.297} C_VEL
LIN {X 0,Y 495.72,Z 276.36,A -85,B 0,C 180,E1 -6171.407,E2 -6171.407} C_VEL
LIN {X 0,Y 495.732,Z 276.359,A -85,B 0,C 180,E1 -6174.462,E2 -6174.462} C_VEL
LIN {X 0,Y 495.765,Z 276.356,A -85,B 0,C 180,E1 -6177.407,E2 -6177.407} C_VEL
LIN {X 0,Y 495.791,Z 276.354,A -85,B 0,C 180,E1 -6180.839,E2 -6180.839} C_VEL
LIN {X 0,Y 499.264,Z 291.188,A -85,B 0,C 180,E1 -6183.228,E2 -6183.228} C_VEL
LIN {X 0,Y 499.379,Z 295.896,A -85,B 0,C 180,E1 -6183.91,E2 -6183.91} C_VEL
LIN {X 0,Y 498.503,Z 316.297,A -85,B 0,C 180,E1 -6186.751,E2 -6186.751} C_VEL
LIN {X 0,Y 498.357,Z 319.918,A -85,B 0,C 180,E1 -6187.249,E2 -6187.249} C_VEL
LIN {X 0,Y 502.102,Z 339.82,A -85,B 0,C 180,E1 -6187.742,E2 -6187.742} C_VEL
LIN {X 0,Y 500.699,Z 486.394,A -85,B 0,C 180,E1 -6189.929,E2 -6189.929} C_VEL
LIN {X 0,Y 500.247,Z 502.414,A -85,B 0,C 180,E1 -6190.335,E2 -6190.335} C_VEL
LIN {X 0,Y 499.788,Z 517.584,A -85,B 0,C 180,E1 -6190.898,E2 -6190.898} C_VEL
LIN {X 0,Y 499.108,Z 532.62,A -85,B 0,C 180,E1 -6191.636,E2 -6191.636} C_VEL
LIN {X 0,Y 498.489,Z 545.949,A -85,B 0,C 180,E1 -6192.462,E2 -6192.462} C_VEL
LIN {X 0,Y 497.855,Z 559.507,A -85,B 0,C 180,E1 -6193.496,E2 -6193.496} C_VEL
LIN {X 0,Y 497.19,Z 571.841,A -85,B 0,C 180,E1 -6194.631,E2 -6194.631} C_VEL
LIN {X 0,Y 496.599,Z 583.095,A -85,B 0,C 180,E1 -6195.87,E2 -6195.87} C_VEL
LIN {X 0,Y 496.068,Z 594.021,A -85,B 0,C 180,E1 -6197.315,E2 -6197.315} C_VEL
LIN {X 0,Y 495.716,Z 603.114,A -85,B 0,C 180,E1 -6198.759,E2 -6198.759} C_VEL
LIN {X 0,Y 495.383,Z 610.651,A -85,B 0,C 180,E1 -6200.199,E2 -6200.199} C_VEL
LIN {X 0,Y 495.216,Z 617.69,A -85,B 0,C 180,E1 -6201.842,E2 -6201.842} C_VEL
LIN {X 0,Y 495.047,Z 623.594,A -85,B 0,C 180,E1 -6203.6,E2 -6203.6} C_VEL
LIN {X 0,Y 495.002,Z 627.405,A -85,B 0,C 180,E1 -6205.114,E2 -6205.114} C_VEL
LIN {X 0,Y 495.025,Z 630.339,A -85,B 0,C 180,E1 -6206.745,E2 -6206.745} C_VEL
LIN {X 0,Y 494.961,Z 632.09,A -85,B 0,C 180,E1 -6208.373,E2 -6208.373} C_VEL
LIN {X 0,Y 494.896,Z 632.691,A -85,B 0,C 180,E1 -6210,E2 -6210} C_VEL
LIN {X 0,Y 494.961,Z 632.096,A -85,B 0,C 180,E1 -6211.628,E2 -6211.628} C_VEL
LIN {X 0,Y 495.025,Z 630.351,A -85,B 0,C 180,E1 -6213.256,E2 -6213.256} C_VEL
LIN {X 0,Y 495.002,Z 627.428,A -85,B 0,C 180,E1 -6214.887,E2 -6214.887} C_VEL
LIN {X 0,Y 495.08,Z 623.26,A -85,B 0,C 180,E1 -6216.521,E2 -6216.521} C_VEL
LIN {X 0,Y 495.216,Z 617.736,A -85,B 0,C 180,E1 -6218.159,E2 -6218.159} C_VEL
LIN {X 0,Y 495.385,Z 610.703,A -85,B 0,C 180,E1 -6219.802,E2 -6219.802} C_VEL
LIN {X 0,Y 495.72,Z 603.182,A -85,B 0,C 180,E1 -6221.241,E2 -6221.241} C_VEL
LIN {X 0,Y 496.084,Z 594.11,A -85,B 0,C 180,E1 -6222.685,E2 -6222.685} C_VEL
LIN {X 0,Y 496.616,Z 583.201,A -85,B 0,C 180,E1 -6224.13,E2 -6224.13} C_VEL
LIN {X 0,Y 497.189,Z 571.972,A -85,B 0,C 180,E1 -6225.369,E2 -6225.369} C_VEL
LIN {X 0,Y 497.857,Z 559.663,A -85,B 0,C 180,E1 -6226.505,E2 -6226.505} C_VEL
LIN {X 0,Y 498.519,Z 546.118,A -85,B 0,C 180,E1 -6227.538,E2 -6227.538} C_VEL
LIN {X 0,Y 499.148,Z 532.806,A -85,B 0,C 180,E1 -6228.363,E2 -6228.363} C_VEL
LIN {X 0,Y 499.732,Z 518.778,A -85,B 0,C 180,E1 -6229.059,E2 -6229.059} C_VEL
LIN {X 0,Y 500.237,Z 503.694,A -85,B 0,C 180,E1 -6229.63,E2 -6229.63} C_VEL
LIN {X 0,Y 500.658,Z 488.689,A -85,B 0,C 180,E1 -6230.027,E2 -6230.027} C_VEL
LIN {X 0,Y 500.942,Z 460.436,A -85,B 0,C 180,E1 -6230.479,E2 -6230.479} C_VEL
LIN {X 0,Y 502.03,Z 338.869,A -85,B 0,C 180,E1 -6232.277,E2 -6232.277} C_VEL
LIN {X 0,Y 498.364,Z 320.186,A -85,B 0,C 180,E1 -6232.752,E2 -6232.752} C_VEL
LIN {X 0,Y 499.242,Z 301.358,A -85,B 0,C 180,E1 -6235.36,E2 -6235.36} C_VEL
LIN {X 0,Y 499.528,Z 293.032,A -85,B 0,C 180,E1 -6236.532,E2 -6236.532} C_VEL
LIN {X 0,Y 496.822,Z 280.73,A -85,B 0,C 180,E1 -6238.465,E2 -6238.465} C_VEL
LIN {X 0,Y 495.784,Z 276.355,A -85,B 0,C 180,E1 -6239.191,E2 -6239.191} C_VEL
LIN {X 0,Y 495.753,Z 276.359,A -85,B 0,C 180,E1 -6242.595,E2 -6242.595} C_VEL
LIN {X 0,Y 495.741,Z 276.36,A -85,B 0,C 180,E1 -6245.538,E2 -6245.538} C_VEL
LIN {X 0,Y 495.74,Z 276.358,A -85,B 0,C 180,E1 -6248.764,E2 -6248.764} C_VEL
LIN {X 0,Y 495.723,Z 276.361,A -85,B 0,C 180,E1 -6251.784,E2 -6251.784} C_VEL
LIN {X 0,Y 495.736,Z 276.356,A -85,B 0,C 180,E1 -6255.14,E2 -6255.14} C_VEL
LIN {X 0,Y 495.724,Z 276.365,A -85,B 0,C 180,E1 -6258.215,E2 -6258.215} C_VEL
LIN {X 0,Y 495.737,Z 276.353,A -85,B 0,C 180,E1 -6261.235,E2 -6261.235} C_VEL
LIN {X 0,Y 495.726,Z 276.356,A -85,B 0,C 180,E1 -6264.46,E2 -6264.46} C_VEL
LIN {X 0,Y 495.749,Z 276.354,A -85,B 0,C 180,E1 -6267.403,E2 -6267.403} C_VEL
LIN {X 0,Y 495.759,Z 276.356,A -85,B 0,C 180,E1 -6270.252,E2 -6270.252} C_VEL
LIN {X 0,Y 495.734,Z 276.355,A -85,B 0,C 180,E1 -6273.27,E2 -6273.27} C_VEL
LIN {X 0,Y 495.735,Z 276.355,A -85,B 0,C 180,E1 -6276.611,E2 -6276.611} C_VEL
LIN {X 0,Y 495.775,Z 276.354,A -85,B 0,C 180,E1 -6279.323,E2 -6279.323} C_VEL
LIN {X 0,Y 495.775,Z 276.359,A -85,B 0,C 180,E1 -6281.827,E2 -6281.827} C_VEL
LIN {X 0,Y 495.781,Z 276.35,A -85,B 0,C 180,E1 -6285.216,E2 -6285.216} C_VEL
LIN {X 0,Y 495.814,Z 276.337,A -85,B 0,C 180,E1 -6288.553,E2 -6288.553} C_VEL
LIN {X 0,Y 495.802,Z 276.352,A -85,B 0,C 180,E1 -6291.85,E2 -6291.85} C_VEL
LIN {X 0,Y 495.846,Z 276.338,A -85,B 0,C 180,E1 -6294.305,E2 -6294.305} C_VEL
LIN {X 0,Y 495.963,Z 276.321,A -85,B 0,C 180,E1 -6297.562,E2 -6297.562} C_VEL
LIN {X 0,Y 495.957,Z 276.329,A -85,B 0,C 180,E1 -6299.999,E2 -6299.999} C_VEL
LIN {X 0,Y 495.968,Z 276.325,A -85,B 0,C 180,E1 -6302.435,E2 -6302.435} C_VEL
LIN {X 0,Y 495.827,Z 276.335,A -85,B 0,C 180,E1 -6305.693,E2 -6305.693} C_VEL
LIN {X 0,Y 495.766,Z 276.347,A -85,B 0,C 180,E1 -6308.97,E2 -6308.97} C_VEL
LIN {X 0,Y 495.818,Z 276.345,A -85,B 0,C 180,E1 -6312.033,E2 -6312.033} C_VEL
LIN {X 0,Y 495.789,Z 276.341,A -85,B 0,C 180,E1 -6315.623,E2 -6315.623} C_VEL
LIN {X 0,Y 495.755,Z 276.348,A -85,B 0,C 180,E1 -6319.028,E2 -6319.028} C_VEL
LIN {X 0,Y 495.727,Z 276.36,A -85,B 0,C 180,E1 -6321.628,E2 -6321.628} C_VEL
LIN {X 0,Y 495.699,Z 276.356,A -85,B 0,C 180,E1 -6324.276,E2 -6324.276} C_VEL
LIN {X 0,Y 495.717,Z 276.351,A -85,B 0,C 180,E1 -6326.978,E2 -6326.978} C_VEL
LIN {X 0,Y 495.744,Z 276.351,A -85,B 0,C 180,E1 -6330.144,E2 -6330.144} C_VEL
LIN {X 0,Y 495.736,Z 276.36,A -85,B 0,C 180,E1 -6333.236,E2 -6333.236} C_VEL
LIN {X 0,Y 495.695,Z 276.349,A -85,B 0,C 180,E1 -6336.086,E2 -6336.086} C_VEL
LIN {X 0,Y 495.744,Z 276.352,A -85,B 0,C 180,E1 -6338.766,E2 -6338.766} C_VEL
LIN {X 0,Y 495.727,Z 276.356,A -85,B 0,C 180,E1 -6341.781,E2 -6341.781} C_VEL
LIN {X 0,Y 495.72,Z 276.354,A -85,B 0,C 180,E1 -6345.14,E2 -6345.14} C_VEL
LIN {X 0,Y 495.733,Z 276.355,A -85,B 0,C 180,E1 -6348.217,E2 -6348.217} C_VEL
LIN {X 0,Y 495.732,Z 276.354,A -85,B 0,C 180,E1 -6351.407,E2 -6351.407} C_VEL
LIN {X 0,Y 495.731,Z 276.354,A -85,B 0,C 180,E1 -6354.461,E2 -6354.461} C_VEL
LIN {X 0,Y 495.748,Z 276.354,A -85,B 0,C 180,E1 -6357.405,E2 -6357.405} C_VEL
LIN {X 0,Y 495.732,Z 276.353,A -85,B 0,C 180,E1 -6360.701,E2 -6360.701} C_VEL
LIN {X 0,Y 495.072,Z 276.441,A -85,B 0,C 180,E1 -6361.38,E2 -6361.38} C_VEL
LIN {X 0,Y 492.217,Z 276.796,A -85,B 0,C 180,E1 -6362.483,E2 -6362.483} C_VEL
LIN {X 0,Y 489.806,Z 277.094,A -85,B 0,C 180,E1 -6363.372,E2 -6363.372} C_VEL
LIN {X 0,Y 488.781,Z 277.22,A -85,B 0,C 180,E1 -6364.058,E2 -6364.058} C_VEL
LIN {X 0,Y 488.703,Z 277.231,A -85,B 0,C 180,E1 -6364.291,E2 -6364.291} C_VEL
LIN {X 0,Y 488.703,Z 277.236,A -85,B 0,C 180,E1 -6367.152,E2 -6367.152} C_VEL
LIN {X 0,Y 488.706,Z 277.227,A -85,B 0,C 180,E1 -6369.81,E2 -6369.81} C_VEL
LIN {X 0,Y 488.71,Z 277.235,A -85,B 0,C 180,E1 -6372.423,E2 -6372.423} C_VEL
LIN {X 0,Y 488.742,Z 277.231,A -85,B 0,C 180,E1 -6374.999,E2 -6374.999} C_VEL
LIN {X 0,Y 488.814,Z 277.222,A -85,B 0,C 180,E1 -6378.388,E2 -6378.388} C_VEL
LIN {X 0,Y 488.797,Z 277.219,A -85,B 0,C 180,E1 -6381.733,E2 -6381.733} C_VEL
LIN {X 0,Y 488.828,Z 277.219,A -85,B 0,C 180,E1 -6384.224,E2 -6384.224} C_VEL
LIN {X 0,Y 488.94,Z 277.204,A -85,B 0,C 180,E1 -6387.528,E2 -6387.528} C_VEL
LIN {X 0,Y 488.947,Z 277.208,A -85,B 0,C 180,E1 -6390,E2 -6390} C_VEL
LIN {X 0,Y 488.941,Z 277.212,A -85,B 0,C 180,E1 -6392.471,E2 -6392.471} C_VEL
LIN {X 0,Y 488.703,Z 277.307,A -85,B 0,C 180,E1 -6393.916,E2 -6393.916} C_VEL
LIN {X 0,Y 491.292,Z 288.575,A -85,B 0,C 180,E1 -6395.953,E2 -6395.953} C_VEL
LIN {X 0,Y 491.749,Z 292.122,A -85,B 0,C 180,E1 -6396.565,E2 -6396.565} C_VEL
LIN {X 0,Y 491.687,Z 295.015,A -85,B 0,C 180,E1 -6397.004,E2 -6397.004} C_VEL
LIN {X 0,Y 495.667,Z 313.3,A -85,B 0,C 180,E1 -6397.485,E2 -6397.485} C_VEL
LIN {X 0,Y 494.159,Z 459.516,A -85,B 0,C 180,E1 -6399.697,E2 -6399.697} C_VEL
LIN {X 0,Y 493.756,Z 475.407,A -85,B 0,C 180,E1 -6400.105,E2 -6400.105} C_VEL
LIN {X 0,Y 493.221,Z 490.619,A -85,B 0,C 180,E1 -6400.675,E2 -6400.675} C_VEL
LIN {X 0,Y 492.647,Z 505.404,A -85,B 0,C 180,E1 -6401.416,E2 -6401.416} C_VEL
LIN {X 0,Y 491.974,Z 518.928,A -85,B 0,C 180,E1 -6402.268,E2 -6402.268} C_VEL
LIN {X 0,Y 491.317,Z 531.396,A -85,B 0,C 180,E1 -6403.23,E2 -6403.23} C_VEL
LIN {X 0,Y 490.59,Z 544.095,A -85,B 0,C 180,E1 -6404.412,E2 -6404.412} C_VEL
LIN {X 0,Y 489.971,Z 554.729,A -85,B 0,C 180,E1 -6405.601,E2 -6405.601} C_VEL
LIN {X 0,Y 489.399,Z 564.596,A -85,B 0,C 180,E1 -6406.905,E2 -6406.905} C_VEL
LIN {X 0,Y 488.9,Z 574.272,A -85,B 0,C 180,E1 -6408.436,E2 -6408.436} C_VEL
LIN {X 0,Y 488.527,Z 582.305,A -85,B 0,C 180,E1 -6409.978,E2 -6409.978} C_VEL
LIN {X 0,Y 488.243,Z 588.941,A -85,B 0,C 180,E1 -6411.534,E2 -6411.534} C_VEL
LIN {X 0,Y 488.076,Z 594.983,A -85,B 0,C 180,E1 -6413.326,E2 -6413.326} C_VEL
LIN {X 0,Y 487.958,Z 598.909,A -85,B 0,C 180,E1 -6414.86,E2 -6414.86} C_VEL
LIN {X 0,Y 487.824,Z 601.986,A -85,B 0,C 180,E1 -6416.525,E2 -6416.525} C_VEL
LIN {X 0,Y 487.811,Z 603.996,A -85,B 0,C 180,E1 -6418.387,E2 -6418.387} C_VEL
LIN {X 0,Y 487.789,Z 604.557,A -85,B 0,C 180,E1 -6420.282,E2 -6420.282} C_VEL
LIN {X 0,Y 487.79,Z 603.964,A -85,B 0,C 180,E1 -6421.786,E2 -6421.786} C_VEL
LIN {X 0,Y 487.814,Z 602.338,A -85,B 0,C 180,E1 -6423.324,E2 -6423.324} C_VEL
LIN {X 0,Y 487.943,Z 599.059,A -85,B 0,C 180,E1 -6425.178,E2 -6425.178} C_VEL
LIN {X 0,Y 488.083,Z 595.219,A -85,B 0,C 180,E1 -6426.698,E2 -6426.698} C_VEL
LIN {X 0,Y 488.229,Z 590.209,A -85,B 0,C 180,E1 -6428.24,E2 -6428.24} C_VEL
LIN {X 0,Y 488.51,Z 583.824,A -85,B 0,C 180,E1 -6429.806,E2 -6429.806} C_VEL
LIN {X 0,Y 488.864,Z 575.823,A -85,B 0,C 180,E1 -6431.398,E2 -6431.398} C_VEL
LIN {X 0,Y 489.292,Z 566.643,A -85,B 0,C 180,E1 -6432.903,E2 -6432.903} C_VEL
LIN {X 0,Y 489.925,Z 556.072,A -85,B 0,C 180,E1 -6434.34,E2 -6434.34} C_VEL
LIN {X 0,Y 490.546,Z 544.604,A -85,B 0,C 180,E1 -6435.638,E2 -6435.638} C_VEL
LIN {X 0,Y 491.3,Z 531.684,A -85,B 0,C 180,E1 -6436.847,E2 -6436.847} C_VEL
LIN {X 0,Y 491.963,Z 519.031,A -85,B 0,C 180,E1 -6437.826,E2 -6437.826} C_VEL
LIN {X 0,Y 492.677,Z 504.67,A -85,B 0,C 180,E1 -6438.726,E2 -6438.726} C_VEL
LIN {X 0,Y 493.308,Z 489.817,A -85,B 0,C 180,E1 -6439.454,E2 -6439.454} C_VEL
LIN {X 0,Y 493.825,Z 474.354,A -85,B 0,C 180,E1 -6440.02,E2 -6440.02} C_VEL
LIN {X 0,Y 494.174,Z 458.68,A -85,B 0,C 180,E1 -6440.411,E2 -6440.411} C_VEL
LIN {X 0,Y 495.654,Z 312.48,A -85,B 0,C 180,E1 -6442.63,E2 -6442.63} C_VEL
LIN {X 0,Y 491.706,Z 295.12,A -85,B 0,C 180,E1 -6443.11,E2 -6443.11} C_VEL
LIN {X 0,Y 491.662,Z 290.476,A -85,B 0,C 180,E1 -6443.884,E2 -6443.884} C_VEL
LIN {X 0,Y 488.698,Z 277.238,A -85,B 0,C 180,E1 -6446.304,E2 -6446.304} C_VEL
LIN {X 0,Y 488.701,Z 277.238,A -85,B 0,C 180,E1 -6449.636,E2 -6449.636} C_VEL
LIN {X 0,Y 488.782,Z 277.226,A -85,B 0,C 180,E1 -6453.056,E2 -6453.056} C_VEL
LIN {X 0,Y 488.677,Z 277.238,A -85,B 0,C 180,E1 -6456.256,E2 -6456.256} C_VEL
LIN {X 0,Y 488.73,Z 277.236,A -85,B 0,C 180,E1 -6459.177,E2 -6459.177} C_VEL
LIN {X 0,Y 488.744,Z 277.232,A -85,B 0,C 180,E1 -6461.629,E2 -6461.629} C_VEL
LIN {X 0,Y 488.747,Z 277.233,A -85,B 0,C 180,E1 -6465.001,E2 -6465.001} C_VEL
LIN {X 0,Y 488.791,Z 277.222,A -85,B 0,C 180,E1 -6468.389,E2 -6468.389} C_VEL
LIN {X 0,Y 488.802,Z 277.22,A -85,B 0,C 180,E1 -6471.735,E2 -6471.735} C_VEL
LIN {X 0,Y 488.833,Z 277.214,A -85,B 0,C 180,E1 -6474.225,E2 -6474.225} C_VEL
LIN {X 0,Y 488.946,Z 277.203,A -85,B 0,C 180,E1 -6477.53,E2 -6477.53} C_VEL
LIN {X 0,Y 488.942,Z 277.208,A -85,B 0,C 180,E1 -6480.825,E2 -6480.825} C_VEL
LIN {X 0,Y 488.945,Z 277.202,A -85,B 0,C 180,E1 -6482.473,E2 -6482.473} C_VEL
LIN {X 0,Y 488.827,Z 277.216,A -85,B 0,C 180,E1 -6485.777,E2 -6485.777} C_VEL
LIN {X 0,Y 488.772,Z 277.222,A -85,B 0,C 180,E1 -6488.268,E2 -6488.268} C_VEL
LIN {X 0,Y 488.794,Z 277.219,A -85,B 0,C 180,E1 -6491.614,E2 -6491.614} C_VEL
LIN {X 0,Y 488.751,Z 277.229,A -85,B 0,C 180,E1 -6495.002,E2 -6495.002} C_VEL
LIN {X 0,Y 488.738,Z 277.232,A -85,B 0,C 180,E1 -6498.444,E2 -6498.444} C_VEL
LIN {X 0,Y 488.698,Z 277.234,A -85,B 0,C 180,E1 -6501.072,E2 -6501.072} C_VEL
LIN {X 0,Y 488.659,Z 277.236,A -85,B 0,C 180,E1 -6503.748,E2 -6503.748} C_VEL
LIN {X 0,Y 488.689,Z 277.235,A -85,B 0,C 180,E1 -6506.923,E2 -6506.923} C_VEL
LIN {X 0,Y 488.699,Z 277.23,A -85,B 0,C 180,E1 -6509.273,E2 -6509.273} C_VEL
LIN {X 0,Y 488.687,Z 277.236,A -85,B 0,C 180,E1 -6512.149,E2 -6512.149} C_VEL
LIN {X 0,Y 488.698,Z 277.232,A -85,B 0,C 180,E1 -6515.118,E2 -6515.118} C_VEL
LIN {X 0,Y 488.647,Z 277.245,A -85,B 0,C 180,E1 -6518.204,E2 -6518.204} C_VEL
LIN {X 0,Y 488.688,Z 277.239,A -85,B 0,C 180,E1 -6520.342,E2 -6520.342} C_VEL
LIN {X 0,Y 488.667,Z 277.238,A -85,B 0,C 180,E1 -6523.657,E2 -6523.657} C_VEL
LIN {X 0,Y 488.66,Z 277.242,A -85,B 0,C 180,E1 -6526.344,E2 -6526.344} C_VEL
LIN {X 0,Y 488.7,Z 277.236,A -85,B 0,C 180,E1 -6529.675,E2 -6529.675} C_VEL
LIN {X 0,Y 488.648,Z 277.236,A -85,B 0,C 180,E1 -6532.84,E2 -6532.84} C_VEL
LIN {X 0,Y 488.721,Z 277.233,A -85,B 0,C 180,E1 -6535.888,E2 -6535.888} C_VEL
LIN {X 0,Y 488.689,Z 277.236,A -85,B 0,C 180,E1 -6538.821,E2 -6538.821} C_VEL
LIN {X 0,Y 488.727,Z 277.249,A -85,B 0,C 180,E1 -6540.554,E2 -6540.554} C_VEL
LIN {X 0,Y 492.361,Z 292.583,A -85,B 0,C 180,E1 -6543.052,E2 -6543.052} C_VEL
LIN {X 0,Y 492.575,Z 297.294,A -85,B 0,C 180,E1 -6543.75,E2 -6543.75} C_VEL
LIN {X 0,Y 491.537,Z 319.499,A -85,B 0,C 180,E1 -6546.885,E2 -6546.885} C_VEL
LIN {X 0,Y 491.955,Z 322.008,A -85,B 0,C 180,E1 -6546.978,E2 -6546.978} C_VEL
LIN {X 0,Y 495.525,Z 341.081,A -85,B 0,C 180,E1 -6547.453,E2 -6547.453} C_VEL
LIN {X 0,Y 494.015,Z 486.56,A -85,B 0,C 180,E1 -6549.657,E2 -6549.657} C_VEL
LIN {X 0,Y 493.521,Z 502.448,A -85,B 0,C 180,E1 -6550.068,E2 -6550.068} C_VEL
LIN {X 0,Y 493.062,Z 516.664,A -85,B 0,C 180,E1 -6550.599,E2 -6550.599} C_VEL
LIN {X 0,Y 492.425,Z 530.457,A -85,B 0,C 180,E1 -6551.27,E2 -6551.27} C_VEL
LIN {X 0,Y 491.767,Z 544.119,A -85,B 0,C 180,E1 -6552.106,E2 -6552.106} C_VEL
LIN {X 0,Y 491.055,Z 556.693,A -85,B 0,C 180,E1 -6553.047,E2 -6553.047} C_VEL
LIN {X 0,Y 490.387,Z 569.466,A -85,B 0,C 180,E1 -6554.2,E2 -6554.2} C_VEL
LIN {X 0,Y 489.756,Z 581.064,A -85,B 0,C 180,E1 -6555.457,E2 -6555.457} C_VEL
LIN {X 0,Y 489.236,Z 590.825,A -85,B 0,C 180,E1 -6556.713,E2 -6556.713} C_VEL
LIN {X 0,Y 488.771,Z 600.599,A -85,B 0,C 180,E1 -6558.209,E2 -6558.209} C_VEL
LIN {X 0,Y 488.469,Z 608.391,A -85,B 0,C 180,E1 -6559.64,E2 -6559.64} C_VEL
LIN {X 0,Y 488.158,Z 615.84,A -85,B 0,C 180,E1 -6561.306,E2 -6561.306} C_VEL
LIN {X 0,Y 488.05,Z 621.752,A -85,B 0,C 180,E1 -6562.97,E2 -6562.97} C_VEL
LIN {X 0,Y 487.963,Z 625.264,A -85,B 0,C 180,E1 -6564.214,E2 -6564.214} C_VEL
LIN {X 0,Y 487.879,Z 628.815,A -85,B 0,C 180,E1 -6565.87,E2 -6565.87} C_VEL
LIN {X 0,Y 487.905,Z 631.154,A -85,B 0,C 180,E1 -6567.524,E2 -6567.524} C_VEL
LIN {X 0,Y 487.832,Z 632.332,A -85,B 0,C 180,E1 -6569.175,E2 -6569.175} C_VEL
LIN {X 0,Y 487.832,Z 632.336,A -85,B 0,C 180,E1 -6570.826,E2 -6570.826} C_VEL
LIN {X 0,Y 487.905,Z 631.166,A -85,B 0,C 180,E1 -6572.477,E2 -6572.477} C_VEL
LIN {X 0,Y 487.879,Z 628.836,A -85,B 0,C 180,E1 -6574.131,E2 -6574.131} C_VEL
LIN {X 0,Y 487.965,Z 625.302,A -85,B 0,C 180,E1 -6575.787,E2 -6575.787} C_VEL
LIN {X 0,Y 488.066,Z 620.469,A -85,B 0,C 180,E1 -6577.446,E2 -6577.446} C_VEL
LIN {X 0,Y 488.229,Z 614.209,A -85,B 0,C 180,E1 -6579.111,E2 -6579.111} C_VEL
LIN {X 0,Y 488.587,Z 606.348,A -85,B 0,C 180,E1 -6580.778,E2 -6580.778} C_VEL
LIN {X 0,Y 488.908,Z 597.656,A -85,B 0,C 180,E1 -6582.292,E2 -6582.292} C_VEL
LIN {X 0,Y 489.418,Z 587.902,A -85,B 0,C 180,E1 -6583.706,E2 -6583.706} C_VEL
LIN {X 0,Y 489.902,Z 577.602,A -85,B 0,C 180,E1 -6584.965,E2 -6584.965} C_VEL
LIN {X 0,Y 490.673,Z 564.997,A -85,B 0,C 180,E1 -6586.248,E2 -6586.248} C_VEL
LIN {X 0,Y 491.344,Z 551.603,A -85,B 0,C 180,E1 -6587.373,E2 -6587.373} C_VEL
LIN {X 0,Y 492.124,Z 537.857,A -85,B 0,C 180,E1 -6588.311,E2 -6588.311} C_VEL
LIN {X 0,Y 492.774,Z 523.589,A -85,B 0,C 180,E1 -6589.095,E2 -6589.095} C_VEL
LIN {X 0,Y 493.385,Z 508.573,A -85,B 0,C 180,E1 -6589.73,E2 -6589.73} C_VEL
LIN {X 0,Y 493.865,Z 493.314,A -85,B 0,C 180,E1 -6590.195,E2 -6590.195} C_VEL
LIN {X 0,Y 494.125,Z 477.74,A -85,B 0,C 180,E1 -6590.502,E2 -6590.502} C_VEL
LIN {X 0,Y 495.505,Z 341.05,A -85,B 0,C 180,E1 -6592.549,E2 -6592.549} C_VEL
LIN {X 0,Y 491.559,Z 320.108,A -85,B 0,C 180,E1 -6593.068,E2 -6593.068} C_VEL
LIN {X 0,Y 492.463,Z 301.638,A -85,B 0,C 180,E1 -6595.664,E2 -6595.664} C_VEL
LIN {X 0,Y 492.654,Z 294.398,A -85,B 0,C 180,E1 -6596.703,E2 -6596.703} C_VEL
LIN {X 0,Y 489.604,Z 280.807,A -85,B 0,C 180,E1 -6598.881,E2 -6598.881} C_VEL
LIN {X 0,Y 488.734,Z 277.229,A -85,B 0,C 180,E1 -6599.506,E2 -6599.506} C_VEL
LIN {X 0,Y 488.698,Z 277.238,A -85,B 0,C 180,E1 -6602.147,E2 -6602.147} C_VEL
LIN {X 0,Y 488.712,Z 277.234,A -85,B 0,C 180,E1 -6605.115,E2 -6605.115} C_VEL
LIN {X 0,Y 488.658,Z 277.243,A -85,B 0,C 180,E1 -6608.201,E2 -6608.201} C_VEL
LIN {X 0,Y 488.693,Z 277.236,A -85,B 0,C 180,E1 -6610.34,E2 -6610.34} C_VEL
LIN {X 0,Y 488.672,Z 277.236,A -85,B 0,C 180,E1 -6613.655,E2 -6613.655} C_VEL
LIN {X 0,Y 488.674,Z 277.237,A -85,B 0,C 180,E1 -6616.343,E2 -6616.343} C_VEL
LIN {X 0,Y 488.702,Z 277.238,A -85,B 0,C 180,E1 -6619.673,E2 -6619.673} C_VEL
LIN {X 0,Y 488.646,Z 277.241,A -85,B 0,C 180,E1 -6622.837,E2 -6622.837} C_VEL
LIN {X 0,Y 488.714,Z 277.231,A -85,B 0,C 180,E1 -6625.885,E2 -6625.885} C_VEL
LIN {X 0,Y 488.687,Z 277.233,A -85,B 0,C 180,E1 -6628.819,E2 -6628.819} C_VEL
LIN {X 0,Y 488.694,Z 277.238,A -85,B 0,C 180,E1 -6631.667,E2 -6631.667} C_VEL
LIN {X 0,Y 488.693,Z 277.234,A -85,B 0,C 180,E1 -6634.959,E2 -6634.959} C_VEL
LIN {X 0,Y 488.694,Z 277.239,A -85,B 0,C 180,E1 -6638.042,E2 -6638.042} C_VEL
LIN {X 0,Y 488.73,Z 277.227,A -85,B 0,C 180,E1 -6640.685,E2 -6640.685} C_VEL
LIN {X 0,Y 488.752,Z 277.226,A -85,B 0,C 180,E1 -6644.144,E2 -6644.144} C_VEL
LIN {X 0,Y 488.732,Z 277.219,A -85,B 0,C 180,E1 -6647.542,E2 -6647.542} C_VEL
LIN {X 0,Y 488.719,Z 277.23,A -85,B 0,C 180,E1 -6650.062,E2 -6650.062} C_VEL
LIN {X 0,Y 488.813,Z 277.217,A -85,B 0,C 180,E1 -6652.768,E2 -6652.768} C_VEL
LIN {X 0,Y 488.779,Z 277.219,A -85,B 0,C 180,E1 -6655.05,E2 -6655.05} C_VEL
LIN {X 0,Y 488.929,Z 277.196,A -85,B 0,C 180,E1 -6657.527,E2 -6657.527} C_VEL
LIN {X 0,Y 488.927,Z 277.205,A -85,B 0,C 180,E1 -6659.999,E2 -6659.999} C_VEL
LIN {X 0,Y 488.936,Z 277.201,A -85,B 0,C 180,E1 -6662.47,E2 -6662.47} C_VEL
LIN {X 0,Y 488.784,Z 277.21,A -85,B 0,C 180,E1 -6665.775,E2 -6665.775} C_VEL
LIN {X 0,Y 488.717,Z 277.226,A -85,B 0,C 180,E1 -6669.1,E2 -6669.1} C_VEL
LIN {X 0,Y 488.779,Z 277.222,A -85,B 0,C 180,E1 -6672.113,E2 -6672.113} C_VEL
LIN {X 0,Y 488.764,Z 277.216,A -85,B 0,C 180,E1 -6675.552,E2 -6675.552} C_VEL
LIN {X 0,Y 488.732,Z 277.218,A -85,B 0,C 180,E1 -6678.441,E2 -6678.441} C_VEL
LIN {X 0,Y 488.694,Z 277.235,A -85,B 0,C 180,E1 -6681.069,E2 -6681.069} C_VEL
LIN {X 0,Y 488.655,Z 277.236,A -85,B 0,C 180,E1 -6683.745,E2 -6683.745} C_VEL
LIN {X 0,Y 488.684,Z 277.226,A -85,B 0,C 180,E1 -6686.92,E2 -6686.92} C_VEL
LIN {X 0,Y 488.703,Z 277.228,A -85,B 0,C 180,E1 -6690.218,E2 -6690.218} C_VEL
LIN {X 0,Y 488.695,Z 277.233,A -85,B 0,C 180,E1 -6693.478,E2 -6693.478} C_VEL
LIN {X 0,Y 488.657,Z 277.226,A -85,B 0,C 180,E1 -6696.352,E2 -6696.352} C_VEL
LIN {X 0,Y 488.68,Z 277.239,A -85,B 0,C 180,E1 -6699.254,E2 -6699.254} C_VEL
LIN {X 0,Y 488.651,Z 277.239,A -85,B 0,C 180,E1 -6702.527,E2 -6702.527} C_VEL
LIN {X 0,Y 488.684,Z 277.23,A -85,B 0,C 180,E1 -6705.196,E2 -6705.196} C_VEL
LIN {X 0,Y 488.677,Z 277.237,A -85,B 0,C 180,E1 -6708.582,E2 -6708.582} C_VEL
LIN {X 0,Y 488.686,Z 277.239,A -85,B 0,C 180,E1 -6710.946,E2 -6710.946} C_VEL
LIN {X 0,Y 488.66,Z 277.232,A -85,B 0,C 180,E1 -6713.867,E2 -6713.867} C_VEL
LIN {X 0,Y 488.718,Z 277.238,A -85,B 0,C 180,E1 -6716.876,E2 -6716.876} C_VEL
LIN {X 0,Y 488.704,Z 277.225,A -85,B 0,C 180,E1 -6719.78,E2 -6719.78} C_VEL
LIN {X 0,Y 488.773,Z 277.226,A -85,B 0,C 180,E1 -6723.056,E2 -6723.056} C_VEL
LIN {X 0,Y 488.703,Z 277.231,A -85,B 0,C 180,E1 -6724.291,E2 -6724.291} C_VEL
LIN {X 0,Y 488.05,Z 277.316,A -85,B 0,C 180,E1 -6724.978,E2 -6724.978} C_VEL
LIN {X 0,Y 485.192,Z 277.672,A -85,B 0,C 180,E1 -6726.095,E2 -6726.095} C_VEL
LIN {X 0,Y 482.76,Z 277.978,A -85,B 0,C 180,E1 -6726.995,E2 -6726.995} C_VEL
LIN {X 0,Y 481.707,Z 278.104,A -85,B 0,C 180,E1 -6727.69,E2 -6727.69} C_VEL
LIN {X 0,Y 481.618,Z 278.115,A -85,B 0,C 180,E1 -6727.925,E2 -6727.925} C_VEL
LIN {X 0,Y 481.687,Z 278.105,A -85,B 0,C 180,E1 -6730.392,E2 -6730.392} C_VEL
LIN {X 0,Y 481.669,Z 278.109,A -85,B 0,C 180,E1 -6733.033,E2 -6733.033} C_VEL
LIN {X 0,Y 481.669,Z 278.107,A -85,B 0,C 180,E1 -6735.638,E2 -6735.638} C_VEL
LIN {X 0,Y 481.778,Z 278.097,A -85,B 0,C 180,E1 -6738.216,E2 -6738.216} C_VEL
LIN {X 0,Y 481.743,Z 278.098,A -85,B 0,C 180,E1 -6741.611,E2 -6741.611} C_VEL
LIN {X 0,Y 481.788,Z 278.096,A -85,B 0,C 180,E1 -6744.139,E2 -6744.139} C_VEL
LIN {X 0,Y 481.908,Z 278.081,A -85,B 0,C 180,E1 -6747.492,E2 -6747.492} C_VEL
LIN {X 0,Y 481.919,Z 278.084,A -85,B 0,C 180,E1 -6750,E2 -6750} C_VEL
LIN {X 0,Y 481.908,Z 278.088,A -85,B 0,C 180,E1 -6752.507,E2 -6752.507} C_VEL
LIN {X 0,Y 481.729,Z 278.318,A -85,B 0,C 180,E1 -6753.659,E2 -6753.659} C_VEL
LIN {X 0,Y 484.432,Z 290.155,A -85,B 0,C 180,E1 -6755.828,E2 -6755.828} C_VEL
LIN {X 0,Y 484.875,Z 294.339,A -85,B 0,C 180,E1 -6756.554,E2 -6756.554} C_VEL
LIN {X 0,Y 484.846,Z 294.981,A -85,B 0,C 180,E1 -6756.659,E2 -6756.659} C_VEL
LIN {X 0,Y 489.115,Z 313.945,A -85,B 0,C 180,E1 -6757.177,E2 -6757.177} C_VEL
LIN {X 0,Y 487.514,Z 459.664,A -85,B 0,C 180,E1 -6759.411,E2 -6759.411} C_VEL
LIN {X 0,Y 487.076,Z 475.244,A -85,B 0,C 180,E1 -6759.813,E2 -6759.813} C_VEL
LIN {X 0,Y 486.491,Z 491.162,A -85,B 0,C 180,E1 -6760.418,E2 -6760.418} C_VEL
LIN {X 0,Y 485.89,Z 505.63,A -85,B 0,C 180,E1 -6761.154,E2 -6761.154} C_VEL
LIN {X 0,Y 485.189,Z 519.145,A -85,B 0,C 180,E1 -6762.018,E2 -6762.018} C_VEL
LIN {X 0,Y 484.427,Z 532.852,A -85,B 0,C 180,E1 -6763.101,E2 -6763.101} C_VEL
LIN {X 0,Y 483.646,Z 545.341,A -85,B 0,C 180,E1 -6764.301,E2 -6764.301} C_VEL
LIN {X 0,Y 482.954,Z 556.714,A -85,B 0,C 180,E1 -6765.617,E2 -6765.617} C_VEL
LIN {X 0,Y 482.378,Z 566.343,A -85,B 0,C 180,E1 -6766.94,E2 -6766.94} C_VEL
LIN {X 0,Y 481.831,Z 576.05,A -85,B 0,C 180,E1 -6768.55,E2 -6768.55} C_VEL
LIN {X 0,Y 481.463,Z 583.581,A -85,B 0,C 180,E1 -6770.061,E2 -6770.061} C_VEL
LIN {X 0,Y 481.128,Z 590.846,A -85,B 0,C 180,E1 -6771.868,E2 -6771.868} C_VEL
LIN {X 0,Y 481.016,Z 595.191,A -85,B 0,C 180,E1 -6773.233,E2 -6773.233} C_VEL
LIN {X 0,Y 480.863,Z 599.724,A -85,B 0,C 180,E1 -6775.077,E2 -6775.077} C_VEL
LIN {X 0,Y 480.712,Z 602.819,A -85,B 0,C 180,E1 -6776.949,E2 -6776.949} C_VEL
LIN {X 0,Y 480.694,Z 604.475,A -85,B 0,C 180,E1 -6778.846,E2 -6778.846} C_VEL
LIN {X 0,Y 480.7,Z 604.669,A -85,B 0,C 180,E1 -6780.777,E2 -6780.777} C_VEL
LIN {X 0,Y 480.705,Z 604.018,A -85,B 0,C 180,E1 -6782.013,E2 -6782.013} C_VEL
LIN {X 0,Y 480.729,Z 602.045,A -85,B 0,C 180,E1 -6783.747,E2 -6783.747} C_VEL
LIN {X 0,Y 480.849,Z 599.646,A -85,B 0,C 180,E1 -6785.071,E2 -6785.071} C_VEL
LIN {X 0,Y 481.021,Z 595.407,A -85,B 0,C 180,E1 -6786.799,E2 -6786.799} C_VEL
LIN {X 0,Y 481.186,Z 590.344,A -85,B 0,C 180,E1 -6788.378,E2 -6788.378} C_VEL
LIN {X 0,Y 481.495,Z 583.987,A -85,B 0,C 180,E1 -6789.957,E2 -6789.957} C_VEL
LIN {X 0,Y 481.921,Z 575.126,A -85,B 0,C 180,E1 -6791.724,E2 -6791.724} C_VEL
LIN {X 0,Y 482.432,Z 565.754,A -85,B 0,C 180,E1 -6793.251,E2 -6793.251} C_VEL
LIN {X 0,Y 483.073,Z 555.102,A -85,B 0,C 180,E1 -6794.69,E2 -6794.69} C_VEL
LIN {X 0,Y 483.774,Z 543.47,A -85,B 0,C 180,E1 -6795.998,E2 -6795.998} C_VEL
LIN {X 0,Y 484.472,Z 531.861,A -85,B 0,C 180,E1 -6797.091,E2 -6797.091} C_VEL
LIN {X 0,Y 485.225,Z 518.749,A -85,B 0,C 180,E1 -6798.114,E2 -6798.114} C_VEL
LIN {X 0,Y 485.939,Z 505.249,A -85,B 0,C 180,E1 -6798.971,E2 -6798.971} C_VEL
LIN {X 0,Y 486.585,Z 491.155,A -85,B 0,C 180,E1 -6799.68,E2 -6799.68} C_VEL
LIN {X 0,Y 487.128,Z 476.099,A -85,B 0,C 180,E1 -6800.255,E2 -6800.255} C_VEL
LIN {X 0,Y 487.5,Z 460.481,A -85,B 0,C 180,E1 -6800.67,E2 -6800.67} C_VEL
LIN {X 0,Y 489.14,Z 313.488,A -85,B 0,C 180,E1 -6802.939,E2 -6802.939} C_VEL
LIN {X 0,Y 484.929,Z 295.249,A -85,B 0,C 180,E1 -6803.47,E2 -6803.47} C_VEL
LIN {X 0,Y 484.78,Z 291.87,A -85,B 0,C 180,E1 -6804.049,E2 -6804.049} C_VEL
LIN {X 0,Y 481.685,Z 278.112,A -85,B 0,C 180,E1 -6806.644,E2 -6806.644} C_VEL
LIN {X 0,Y 481.671,Z 278.112,A -85,B 0,C 180,E1 -6810.261,E2 -6810.261} C_VEL
LIN {X 0,Y 481.735,Z 278.104,A -85,B 0,C 180,E1 -6813.114,E2 -6813.114} C_VEL
LIN {X 0,Y 481.661,Z 278.114,A -85,B 0,C 180,E1 -6815.888,E2 -6815.888} C_VEL
LIN {X 0,Y 481.686,Z 278.111,A -85,B 0,C 180,E1 -6819.029,E2 -6819.029} C_VEL
LIN {X 0,Y 481.692,Z 278.107,A -85,B 0,C 180,E1 -6822.16,E2 -6822.16} C_VEL
LIN {X 0,Y 481.727,Z 278.105,A -85,B 0,C 180,E1 -6824.777,E2 -6824.777} C_VEL
LIN {X 0,Y 481.736,Z 278.1,A -85,B 0,C 180,E1 -6828.216,E2 -6828.216} C_VEL
LIN {X 0,Y 481.747,Z 278.1,A -85,B 0,C 180,E1 -6831.613,E2 -6831.613} C_VEL
LIN {X 0,Y 481.794,Z 278.09,A -85,B 0,C 180,E1 -6834.141,E2 -6834.141} C_VEL
LIN {X 0,Y 481.913,Z 278.08,A -85,B 0,C 180,E1 -6837.494,E2 -6837.494} C_VEL
LIN {X 0,Y 481.893,Z 278.087,A -85,B 0,C 180,E1 -6840.837,E2 -6840.837} C_VEL
LIN {X 0,Y 481.912,Z 278.078,A -85,B 0,C 180,E1 -6842.509,E2 -6842.509} C_VEL
LIN {X 0,Y 481.788,Z 278.093,A -85,B 0,C 180,E1 -6845.862,E2 -6845.862} C_VEL
LIN {X 0,Y 481.727,Z 278.101,A -85,B 0,C 180,E1 -6848.39,E2 -6848.39} C_VEL
LIN {X 0,Y 481.74,Z 278.098,A -85,B 0,C 180,E1 -6851.786,E2 -6851.786} C_VEL
LIN {X 0,Y 481.732,Z 278.101,A -85,B 0,C 180,E1 -6855.226,E2 -6855.226} C_VEL
LIN {X 0,Y 481.699,Z 278.109,A -85,B 0,C 180,E1 -6858.723,E2 -6858.723} C_VEL
LIN {X 0,Y 481.636,Z 278.112,A -85,B 0,C 180,E1 -6861.396,E2 -6861.396} C_VEL
LIN {X 0,Y 481.638,Z 278.113,A -85,B 0,C 180,E1 -6864.116,E2 -6864.116} C_VEL
LIN {X 0,Y 481.664,Z 278.109,A -85,B 0,C 180,E1 -6867.123,E2 -6867.123} C_VEL
LIN {X 0,Y 481.66,Z 278.108,A -85,B 0,C 180,E1 -6869.743,E2 -6869.743} C_VEL
LIN {X 0,Y 481.643,Z 278.114,A -85,B 0,C 180,E1 -6872.677,E2 -6872.677} C_VEL
LIN {X 0,Y 481.641,Z 278.111,A -85,B 0,C 180,E1 -6875.203,E2 -6875.203} C_VEL
LIN {X 0,Y 481.622,Z 278.117,A -85,B 0,C 180,E1 -6878.004,E2 -6878.004} C_VEL
LIN {X 0,Y 481.615,Z 278.113,A -85,B 0,C 180,E1 -6881.047,E2 -6881.047} C_VEL
LIN {X 0,Y 481.648,Z 278.115,A -85,B 0,C 180,E1 -6884.46,E2 -6884.46} C_VEL
LIN {X 0,Y 481.61,Z 278.12,A -85,B 0,C 180,E1 -6887.837,E2 -6887.837} C_VEL
LIN {X 0,Y 481.645,Z 278.113,A -85,B 0,C 180,E1 -6890.657,E2 -6890.657} C_VEL
LIN {X 0,Y 481.607,Z 278.114,A -85,B 0,C 180,E1 -6893.38,E2 -6893.38} C_VEL
LIN {X 0,Y 481.675,Z 278.112,A -85,B 0,C 180,E1 -6896.329,E2 -6896.329} C_VEL
LIN {X 0,Y 481.69,Z 278.112,A -85,B 0,C 180,E1 -6899.778,E2 -6899.778} C_VEL
LIN {X 0,Y 481.71,Z 278.275,A -85,B 0,C 180,E1 -6900.262,E2 -6900.262} C_VEL
LIN {X 0,Y 485.442,Z 293.979,A -85,B 0,C 180,E1 -6902.869,E2 -6902.869} C_VEL
LIN {X 0,Y 485.818,Z 297.12,A -85,B 0,C 180,E1 -6903.356,E2 -6903.356} C_VEL
LIN {X 0,Y 484.921,Z 315.91,A -85,B 0,C 180,E1 -6906.059,E2 -6906.059} C_VEL
LIN {X 0,Y 484.71,Z 319.498,A -85,B 0,C 180,E1 -6906.569,E2 -6906.569} C_VEL
LIN {X 0,Y 488.972,Z 341.748,A -85,B 0,C 180,E1 -6907.144,E2 -6907.144} C_VEL
LIN {X 0,Y 487.358,Z 486.242,A -85,B 0,C 180,E1 -6909.366,E2 -6909.366} C_VEL
LIN {X 0,Y 486.824,Z 502.326,A -85,B 0,C 180,E1 -6909.788,E2 -6909.788} C_VEL
LIN {X 0,Y 486.337,Z 516.811,A -85,B 0,C 180,E1 -6910.338,E2 -6910.338} C_VEL
LIN {X 0,Y 485.679,Z 530.193,A -85,B 0,C 180,E1 -6911,E2 -6911} C_VEL
LIN {X 0,Y 484.982,Z 543.859,A -85,B 0,C 180,E1 -6911.847,E2 -6911.847} C_VEL
LIN {X 0,Y 484.221,Z 556.438,A -85,B 0,C 180,E1 -6912.8,E2 -6912.8} C_VEL
LIN {X 0,Y 483.492,Z 569.216,A -85,B 0,C 180,E1 -6913.968,E2 -6913.968} C_VEL
LIN {X 0,Y 482.785,Z 580.821,A -85,B 0,C 180,E1 -6915.242,E2 -6915.242} C_VEL
LIN {X 0,Y 482.243,Z 590.589,A -85,B 0,C 180,E1 -6916.516,E2 -6916.516} C_VEL
LIN {X 0,Y 481.767,Z 599.908,A -85,B 0,C 180,E1 -6917.956,E2 -6917.956} C_VEL
LIN {X 0,Y 481.439,Z 608.167,A -85,B 0,C 180,E1 -6919.487,E2 -6919.487} C_VEL
LIN {X 0,Y 481.096,Z 615.621,A -85,B 0,C 180,E1 -6921.177,E2 -6921.177} C_VEL
LIN {X 0,Y 480.976,Z 621.538,A -85,B 0,C 180,E1 -6922.866,E2 -6922.866} C_VEL
LIN {X 0,Y 480.865,Z 625.052,A -85,B 0,C 180,E1 -6924.128,E2 -6924.128} C_VEL
LIN {X 0,Y 480.784,Z 628.607,A -85,B 0,C 180,E1 -6925.809,E2 -6925.809} C_VEL
LIN {X 0,Y 480.819,Z 630.949,A -85,B 0,C 180,E1 -6927.487,E2 -6927.487} C_VEL
LIN {X 0,Y 480.758,Z 632.129,A -85,B 0,C 180,E1 -6929.163,E2 -6929.163} C_VEL
LIN {X 0,Y 480.758,Z 632.135,A -85,B 0,C 180,E1 -6930.838,E2 -6930.838} C_VEL
LIN {X 0,Y 480.819,Z 630.964,A -85,B 0,C 180,E1 -6932.514,E2 -6932.514} C_VEL
LIN {X 0,Y 480.784,Z 628.633,A -85,B 0,C 180,E1 -6934.192,E2 -6934.192} C_VEL
LIN {X 0,Y 480.871,Z 625.097,A -85,B 0,C 180,E1 -6935.872,E2 -6935.872} C_VEL
LIN {X 0,Y 480.99,Z 620.262,A -85,B 0,C 180,E1 -6937.557,E2 -6937.557} C_VEL
LIN {X 0,Y 481.176,Z 613.999,A -85,B 0,C 180,E1 -6939.246,E2 -6939.246} C_VEL
LIN {X 0,Y 481.566,Z 606.134,A -85,B 0,C 180,E1 -6940.937,E2 -6940.937} C_VEL
LIN {X 0,Y 481.85,Z 598.291,A -85,B 0,C 180,E1 -6942.338,E2 -6942.338} C_VEL
LIN {X 0,Y 482.432,Z 587.675,A -85,B 0,C 180,E1 -6943.908,E2 -6943.908} C_VEL
LIN {X 0,Y 482.962,Z 577.369,A -85,B 0,C 180,E1 -6945.185,E2 -6945.185} C_VEL
LIN {X 0,Y 483.686,Z 566.338,A -85,B 0,C 180,E1 -6946.332,E2 -6946.332} C_VEL
LIN {X 0,Y 484.368,Z 554.022,A -85,B 0,C 180,E1 -6947.413,E2 -6947.413} C_VEL
LIN {X 0,Y 485.188,Z 540.862,A -85,B 0,C 180,E1 -6948.364,E2 -6948.364} C_VEL
LIN {X 0,Y 485.82,Z 528.385,A -85,B 0,C 180,E1 -6949.105,E2 -6949.105} C_VEL
LIN {X 0,Y 486.44,Z 513.831,A -85,B 0,C 180,E1 -6949.794,E2 -6949.794} C_VEL
LIN {X 0,Y 486.993,Z 498.907,A -85,B 0,C 180,E1 -6950.319,E2 -6950.319} C_VEL
LIN {X 0,Y 487.404,Z 483.459,A -85,B 0,C 180,E1 -6950.687,E2 -6950.687} C_VEL
LIN {X 0,Y 488.939,Z 341.725,A -85,B 0,C 180,E1 -6952.853,E2 -6952.853} C_VEL
LIN {X 0,Y 484.744,Z 319.826,A -85,B 0,C 180,E1 -6953.421,E2 -6953.421} C_VEL
LIN {X 0,Y 485.759,Z 300.173,A -85,B 0,C 180,E1 -6956.23,E2 -6956.23} C_VEL
LIN {X 0,Y 485.784,Z 295.766,A -85,B 0,C 180,E1 -6956.878,E2 -6956.878} C_VEL
LIN {X 0,Y 482.328,Z 280.801,A -85,B 0,C 180,E1 -6959.324,E2 -6959.324} C_VEL
LIN {X 0,Y 481.683,Z 278.104,A -85,B 0,C 180,E1 -6959.801,E2 -6959.801} C_VEL
LIN {X 0,Y 481.653,Z 278.115,A -85,B 0,C 180,E1 -6962.675,E2 -6962.675} C_VEL
LIN {X 0,Y 481.628,Z 278.119,A -85,B 0,C 180,E1 -6965.71,E2 -6965.71} C_VEL
LIN {X 0,Y 481.632,Z 278.116,A -85,B 0,C 180,E1 -6968.862,E2 -6968.862} C_VEL
LIN {X 0,Y 481.621,Z 278.12,A -85,B 0,C 180,E1 -6971.908,E2 -6971.908} C_VEL
LIN {X 0,Y 481.653,Z 278.114,A -85,B 0,C 180,E1 -6974.457,E2 -6974.457} C_VEL
LIN {X 0,Y 481.624,Z 278.118,A -85,B 0,C 180,E1 -6977.836,E2 -6977.836} C_VEL
LIN {X 0,Y 481.647,Z 278.109,A -85,B 0,C 180,E1 -6980.655,E2 -6980.655} C_VEL
LIN {X 0,Y 481.605,Z 278.12,A -85,B 0,C 180,E1 -6983.379,E2 -6983.379} C_VEL
LIN {X 0,Y 481.668,Z 278.109,A -85,B 0,C 180,E1 -6986.326,E2 -6986.326} C_VEL
LIN {X 0,Y 481.646,Z 278.112,A -85,B 0,C 180,E1 -6989.417,E2 -6989.417} C_VEL
LIN {X 0,Y 481.648,Z 278.112,A -85,B 0,C 180,E1 -6992.164,E2 -6992.164} C_VEL
LIN {X 0,Y 481.667,Z 278.109,A -85,B 0,C 180,E1 -6994.966,E2 -6994.966} C_VEL
LIN {X 0,Y 481.644,Z 278.117,A -85,B 0,C 180,E1 -6997.703,E2 -6997.703} C_VEL
LIN {X 0,Y 481.695,Z 278.104,A -85,B 0,C 180,E1 -7000.392,E2 -7000.392} C_VEL
LIN {X 0,Y 481.66,Z 278.111,A -85,B 0,C 180,E1 -7003.032,E2 -7003.032} C_VEL
LIN {X 0,Y 481.679,Z 278.104,A -85,B 0,C 180,E1 -7005.637,E2 -7005.637} C_VEL
LIN {X 0,Y 481.728,Z 278.093,A -85,B 0,C 180,E1 -7008.213,E2 -7008.213} C_VEL
LIN {X 0,Y 481.705,Z 278.109,A -85,B 0,C 180,E1 -7011.609,E2 -7011.609} C_VEL
LIN {X 0,Y 481.767,Z 278.092,A -85,B 0,C 180,E1 -7014.138,E2 -7014.138} C_VEL
LIN {X 0,Y 481.895,Z 278.071,A -85,B 0,C 180,E1 -7017.491,E2 -7017.491} C_VEL
LIN {X 0,Y 481.897,Z 278.08,A -85,B 0,C 180,E1 -7019.999,E2 -7019.999} C_VEL
LIN {X 0,Y 481.903,Z 278.077,A -85,B 0,C 180,E1 -7022.506,E2 -7022.506} C_VEL
LIN {X 0,Y 481.744,Z 278.085,A -85,B 0,C 180,E1 -7025.86,E2 -7025.86} C_VEL
LIN {X 0,Y 481.684,Z 278.104,A -85,B 0,C 180,E1 -7029.234,E2 -7029.234} C_VEL
LIN {X 0,Y 481.743,Z 278.098,A -85,B 0,C 180,E1 -7032.197,E2 -7032.197} C_VEL
LIN {X 0,Y 481.712,Z 278.092,A -85,B 0,C 180,E1 -7035.656,E2 -7035.656} C_VEL
LIN {X 0,Y 481.693,Z 278.096,A -85,B 0,C 180,E1 -7038.721,E2 -7038.721} C_VEL
LIN {X 0,Y 481.632,Z 278.119,A -85,B 0,C 180,E1 -7041.393,E2 -7041.393} C_VEL
LIN {X 0,Y 481.634,Z 278.108,A -85,B 0,C 180,E1 -7044.113,E2 -7044.113} C_VEL
LIN {X 0,Y 481.639,Z 278.102,A -85,B 0,C 180,E1 -7047.116,E2 -7047.116} C_VEL
LIN {X 0,Y 481.651,Z 278.109,A -85,B 0,C 180,E1 -7049.741,E2 -7049.741} C_VEL
LIN {X 0,Y 481.637,Z 278.113,A -85,B 0,C 180,E1 -7052.674,E2 -7052.674} C_VEL
LIN {X 0,Y 481.615,Z 278.104,A -85,B 0,C 180,E1 -7055.709,E2 -7055.709} C_VEL
LIN {X 0,Y 481.651,Z 278.107,A -85,B 0,C 180,E1 -7058.858,E2 -7058.858} C_VEL
LIN {X 0,Y 481.613,Z 278.114,A -85,B 0,C 180,E1 -7062.162,E2 -7062.162} C_VEL
LIN {X 0,Y 481.637,Z 278.106,A -85,B 0,C 180,E1 -7065.541,E2 -7065.541} C_VEL
LIN {X 0,Y 481.632,Z 278.12,A -85,B 0,C 180,E1 -7068.956,E2 -7068.956} C_VEL
LIN {X 0,Y 481.636,Z 278.107,A -85,B 0,C 180,E1 -7071.992,E2 -7071.992} C_VEL
LIN {X 0,Y 481.668,Z 278.111,A -85,B 0,C 180,E1 -7075.317,E2 -7075.317} C_VEL
LIN {X 0,Y 481.626,Z 278.113,A -85,B 0,C 180,E1 -7078.311,E2 -7078.311} C_VEL
LIN {X 0,Y 481.679,Z 278.109,A -85,B 0,C 180,E1 -7081.218,E2 -7081.218} C_VEL
LIN {X 0,Y 481.67,Z 278.105,A -85,B 0,C 180,E1 -7084.041,E2 -7084.041} C_VEL
LIN {X 0,Y 481.656,Z 278.116,A -85,B 0,C 180,E1 -7086.811,E2 -7086.811} C_VEL
LIN {X 0,Y 481.618,Z 278.115,A -85,B 0,C 180,E1 -7087.925,E2 -7087.925} C_VEL
LIN {X 0,Y 480.949,Z 278.204,A -85,B 0,C 180,E1 -7088.624,E2 -7088.624} C_VEL
LIN {X 0,Y 478.125,Z 278.553,A -85,B 0,C 180,E1 -7089.758,E2 -7089.758} C_VEL
LIN {X 0,Y 475.743,Z 278.849,A -85,B 0,C 180,E1 -7090.673,E2 -7090.673} C_VEL
LIN {X 0,Y 474.72,Z 278.976,A -85,B 0,C 180,E1 -7091.378,E2 -7091.378} C_VEL
LIN {X 0,Y 474.637,Z 278.985,A -85,B 0,C 180,E1 -7091.617,E2 -7091.617} C_VEL
LIN {X 0,Y 474.681,Z 278.981,A -85,B 0,C 180,E1 -7094.544,E2 -7094.544} C_VEL
LIN {X 0,Y 474.722,Z 278.974,A -85,B 0,C 180,E1 -7098.038,E2 -7098.038} C_VEL
LIN {X 0,Y 474.709,Z 278.975,A -85,B 0,C 180,E1 -7101.486,E2 -7101.486} C_VEL
LIN {X 0,Y 474.751,Z 278.972,A -85,B 0,C 180,E1 -7104.052,E2 -7104.052} C_VEL
LIN {X 0,Y 474.874,Z 278.957,A -85,B 0,C 180,E1 -7107.455,E2 -7107.455} C_VEL
LIN {X 0,Y 474.89,Z 278.96,A -85,B 0,C 180,E1 -7110,E2 -7110} C_VEL
LIN {X 0,Y 474.743,Z 278.978,A -85,B 0,C 180,E1 -7112.97,E2 -7112.97} C_VEL
LIN {X 0,Y 474.687,Z 279.051,A -85,B 0,C 180,E1 -7113.342,E2 -7113.342} C_VEL
LIN {X 0,Y 477.571,Z 291.728,A -85,B 0,C 180,E1 -7115.7,E2 -7115.7} C_VEL
LIN {X 0,Y 478.083,Z 295.23,A -85,B 0,C 180,E1 -7116.314,E2 -7116.314} C_VEL
LIN {X 0,Y 482.565,Z 314.911,A -85,B 0,C 180,E1 -7116.864,E2 -7116.864} C_VEL
LIN {X 0,Y 480.873,Z 459.781,A -85,B 0,C 180,E1 -7119.118,E2 -7119.118} C_VEL
LIN {X 0,Y 480.414,Z 475.395,A -85,B 0,C 180,E1 -7119.525,E2 -7119.525} C_VEL
LIN {X 0,Y 479.82,Z 490.993,A -85,B 0,C 180,E1 -7120.123,E2 -7120.123} C_VEL
LIN {X 0,Y 479.178,Z 505.554,A -85,B 0,C 180,E1 -7120.869,E2 -7120.869} C_VEL
LIN {X 0,Y 478.409,Z 519.347,A -85,B 0,C 180,E1 -7121.76,E2 -7121.76} C_VEL
LIN {X 0,Y 477.589,Z 532.939,A -85,B 0,C 180,E1 -7122.847,E2 -7122.847} C_VEL
LIN {X 0,Y 476.78,Z 545.554,A -85,B 0,C 180,E1 -7124.076,E2 -7124.076} C_VEL
LIN {X 0,Y 476.024,Z 556.94,A -85,B 0,C 180,E1 -7125.411,E2 -7125.411} C_VEL
LIN {X 0,Y 475.405,Z 566.57,A -85,B 0,C 180,E1 -7126.754,E2 -7126.754} C_VEL
LIN {X 0,Y 474.826,Z 576.263,A -85,B 0,C 180,E1 -7128.385,E2 -7128.385} C_VEL
LIN {X 0,Y 474.442,Z 583.795,A -85,B 0,C 180,E1 -7129.919,E2 -7129.919} C_VEL
LIN {X 0,Y 474.151,Z 589.479,A -85,B 0,C 180,E1 -7131.323,E2 -7131.323} C_VEL
LIN {X 0,Y 473.94,Z 595.492,A -85,B 0,C 180,E1 -7133.169,E2 -7133.169} C_VEL
LIN {X 0,Y 473.823,Z 598.952,A -85,B 0,C 180,E1 -7134.538,E2 -7134.538} C_VEL
LIN {X 0,Y 473.642,Z 602.398,A -85,B 0,C 180,E1 -7136.432,E2 -7136.432} C_VEL
LIN {X 0,Y 473.611,Z 604.405,A -85,B 0,C 180,E1 -7138.349,E2 -7138.349} C_VEL
LIN {X 0,Y 473.613,Z 604.961,A -85,B 0,C 180,E1 -7140.299,E2 -7140.299} C_VEL
LIN {X 0,Y 473.624,Z 604.033,A -85,B 0,C 180,E1 -7142.245,E2 -7142.245} C_VEL
LIN {X 0,Y 473.65,Z 602.237,A -85,B 0,C 180,E1 -7143.81,E2 -7143.81} C_VEL
LIN {X 0,Y 473.843,Z 598.296,A -85,B 0,C 180,E1 -7145.862,E2 -7145.862} C_VEL
LIN {X 0,Y 474.014,Z 594.07,A -85,B 0,C 180,E1 -7147.436,E2 -7147.436} C_VEL
LIN {X 0,Y 474.273,Z 587.534,A -85,B 0,C 180,E1 -7149.307,E2 -7149.307} C_VEL
LIN {X 0,Y 474.667,Z 580.177,A -85,B 0,C 180,E1 -7150.968,E2 -7150.968} C_VEL
LIN {X 0,Y 475.096,Z 571.841,A -85,B 0,C 180,E1 -7152.512,E2 -7152.512} C_VEL
LIN {X 0,Y 475.692,Z 562.324,A -85,B 0,C 180,E1 -7153.977,E2 -7153.977} C_VEL
LIN {X 0,Y 476.398,Z 551.412,A -85,B 0,C 180,E1 -7155.38,E2 -7155.38} C_VEL
LIN {X 0,Y 477.217,Z 539.565,A -85,B 0,C 180,E1 -7156.646,E2 -7156.646} C_VEL
LIN {X 0,Y 477.961,Z 527.401,A -85,B 0,C 180,E1 -7157.73,E2 -7157.73} C_VEL
LIN {X 0,Y 478.686,Z 514.945,A -85,B 0,C 180,E1 -7158.651,E2 -7158.651} C_VEL
LIN {X 0,Y 479.377,Z 501.892,A -85,B 0,C 180,E1 -7159.441,E2 -7159.441} C_VEL
LIN {X 0,Y 480.042,Z 487.182,A -85,B 0,C 180,E1 -7160.142,E2 -7160.142} C_VEL
LIN {X 0,Y 480.591,Z 471.937,A -85,B 0,C 180,E1 -7160.679,E2 -7160.679} C_VEL
LIN {X 0,Y 480.964,Z 456.225,A -85,B 0,C 180,E1 -7161.048,E2 -7161.048} C_VEL
LIN {X 0,Y 482.603,Z 315.191,A -85,B 0,C 180,E1 -7163.246,E2 -7163.246} C_VEL
LIN {X 0,Y 478.729,Z 297.866,A -85,B 0,C 180,E1 -7163.737,E2 -7163.737} C_VEL
LIN {X 0,Y 478.133,Z 295.574,A -85,B 0,C 180,E1 -7163.815,E2 -7163.815} C_VEL
LIN {X 0,Y 477.062,Z 289.446,A -85,B 0,C 180,E1 -7164.935,E2 -7164.935} C_VEL
LIN {X 0,Y 474.649,Z 278.988,A -85,B 0,C 180,E1 -7166.946,E2 -7166.946} C_VEL
LIN {X 0,Y 474.596,Z 278.994,A -85,B 0,C 180,E1 -7169.771,E2 -7169.771} C_VEL
LIN {X 0,Y 474.698,Z 278.979,A -85,B 0,C 180,E1 -7172.682,E2 -7172.682} C_VEL
LIN {X 0,Y 474.643,Z 278.988,A -85,B 0,C 180,E1 -7175.508,E2 -7175.508} C_VEL
LIN {X 0,Y 474.655,Z 278.99,A -85,B 0,C 180,E1 -7179.187,E2 -7179.187} C_VEL
LIN {X 0,Y 474.642,Z 278.987,A -85,B 0,C 180,E1 -7181.886,E2 -7181.886} C_VEL
LIN {X 0,Y 474.685,Z 278.98,A -85,B 0,C 180,E1 -7184.546,E2 -7184.546} C_VEL
LIN {X 0,Y 474.689,Z 278.978,A -85,B 0,C 180,E1 -7188.039,E2 -7188.039} C_VEL
LIN {X 0,Y 474.713,Z 278.977,A -85,B 0,C 180,E1 -7191.488,E2 -7191.488} C_VEL
LIN {X 0,Y 474.756,Z 278.967,A -85,B 0,C 180,E1 -7194.054,E2 -7194.054} C_VEL
LIN {X 0,Y 474.879,Z 278.956,A -85,B 0,C 180,E1 -7197.457,E2 -7197.457} C_VEL
LIN {X 0,Y 474.845,Z 278.965,A -85,B 0,C 180,E1 -7200.849,E2 -7200.849} C_VEL
LIN {X 0,Y 474.878,Z 278.955,A -85,B 0,C 180,E1 -7202.546,E2 -7202.546} C_VEL
LIN {X 0,Y 474.751,Z 278.969,A -85,B 0,C 180,E1 -7205.949,E2 -7205.949} C_VEL
LIN {X 0,Y 474.699,Z 278.978,A -85,B 0,C 180,E1 -7208.515,E2 -7208.515} C_VEL
LIN {X 0,Y 474.694,Z 278.976,A -85,B 0,C 180,E1 -7211.964,E2 -7211.964} C_VEL
LIN {X 0,Y 474.69,Z 278.978,A -85,B 0,C 180,E1 -7215.457,E2 -7215.457} C_VEL
LIN {X 0,Y 474.654,Z 278.983,A -85,B 0,C 180,E1 -7219.012,E2 -7219.012} C_VEL
LIN {X 0,Y 474.579,Z 278.991,A -85,B 0,C 180,E1 -7221.73,E2 -7221.73} C_VEL
LIN {X 0,Y 474.616,Z 278.993,A -85,B 0,C 180,E1 -7224.496,E2 -7224.496} C_VEL
LIN {X 0,Y 474.63,Z 278.984,A -85,B 0,C 180,E1 -7227.325,E2 -7227.325} C_VEL
LIN {X 0,Y 474.588,Z 278.994,A -85,B 0,C 180,E1 -7230.232,E2 -7230.232} C_VEL
LIN {X 0,Y 474.607,Z 278.987,A -85,B 0,C 180,E1 -7233.224,E2 -7233.224} C_VEL
LIN {X 0,Y 474.563,Z 278.996,A -85,B 0,C 180,E1 -7236.327,E2 -7236.327} C_VEL
LIN {X 0,Y 474.593,Z 278.988,A -85,B 0,C 180,E1 -7239.645,E2 -7239.645} C_VEL
LIN {X 0,Y 474.563,Z 278.993,A -85,B 0,C 180,E1 -7242.941,E2 -7242.941} C_VEL
LIN {X 0,Y 474.593,Z 278.993,A -85,B 0,C 180,E1 -7245.895,E2 -7245.895} C_VEL
LIN {X 0,Y 474.587,Z 278.992,A -85,B 0,C 180,E1 -7249.341,E2 -7249.341} C_VEL
LIN {X 0,Y 474.587,Z 278.996,A -85,B 0,C 180,E1 -7251.708,E2 -7251.708} C_VEL
LIN {X 0,Y 474.612,Z 278.989,A -85,B 0,C 180,E1 -7254.726,E2 -7254.726} C_VEL
LIN {X 0,Y 474.633,Z 278.991,A -85,B 0,C 180,E1 -7257.789,E2 -7257.789} C_VEL
LIN {X 0,Y 474.667,Z 279.132,A -85,B 0,C 180,E1 -7259.929,E2 -7259.929} C_VEL
LIN {X 0,Y 478.217,Z 294.005,A -85,B 0,C 180,E1 -7262.451,E2 -7262.451} C_VEL
LIN {X 0,Y 479.008,Z 298.32,A -85,B 0,C 180,E1 -7263.15,E2 -7263.15} C_VEL
LIN {X 0,Y 478.091,Z 316.686,A -85,B 0,C 180,E1 -7265.836,E2 -7265.836} C_VEL
LIN {X 0,Y 477.949,Z 319.25,A -85,B 0,C 180,E1 -7266.206,E2 -7266.206} C_VEL
LIN {X 0,Y 482.438,Z 343.124,A -85,B 0,C 180,E1 -7266.839,E2 -7266.839} C_VEL
LIN {X 0,Y 480.714,Z 485.99,A -85,B 0,C 180,E1 -7269.068,E2 -7269.068} C_VEL
LIN {X 0,Y 480.183,Z 501.892,A -85,B 0,C 180,E1 -7269.489,E2 -7269.489} C_VEL
LIN {X 0,Y 479.611,Z 516.939,A -85,B 0,C 180,E1 -7270.069,E2 -7270.069} C_VEL
LIN {X 0,Y 478.914,Z 529.938,A -85,B 0,C 180,E1 -7270.721,E2 -7270.721} C_VEL
LIN {X 0,Y 478.189,Z 543.612,A -85,B 0,C 180,E1 -7271.58,E2 -7271.58} C_VEL
LIN {X 0,Y 477.368,Z 556.197,A -85,B 0,C 180,E1 -7272.545,E2 -7272.545} C_VEL
LIN {X 0,Y 476.607,Z 568.98,A -85,B 0,C 180,E1 -7273.73,E2 -7273.73} C_VEL
LIN {X 0,Y 475.833,Z 580.585,A -85,B 0,C 180,E1 -7275.021,E2 -7275.021} C_VEL
LIN {X 0,Y 475.26,Z 590.356,A -85,B 0,C 180,E1 -7276.315,E2 -7276.315} C_VEL
LIN {X 0,Y 474.716,Z 599.352,A -85,B 0,C 180,E1 -7277.718,E2 -7277.718} C_VEL
LIN {X 0,Y 474.379,Z 607.943,A -85,B 0,C 180,E1 -7279.328,E2 -7279.328} C_VEL
LIN {X 0,Y 474.042,Z 615.403,A -85,B 0,C 180,E1 -7281.045,E2 -7281.045} C_VEL
LIN {X 0,Y 473.901,Z 621.324,A -85,B 0,C 180,E1 -7282.759,E2 -7282.759} C_VEL
LIN {X 0,Y 473.771,Z 624.84,A -85,B 0,C 180,E1 -7284.04,E2 -7284.04} C_VEL
LIN {X 0,Y 473.693,Z 628.399,A -85,B 0,C 180,E1 -7285.746,E2 -7285.746} C_VEL
LIN {X 0,Y 473.736,Z 630.745,A -85,B 0,C 180,E1 -7287.45,E2 -7287.45} C_VEL
LIN {X 0,Y 473.686,Z 631.926,A -85,B 0,C 180,E1 -7289.15,E2 -7289.15} C_VEL
LIN {X 0,Y 473.687,Z 631.933,A -85,B 0,C 180,E1 -7290.85,E2 -7290.85} C_VEL
LIN {X 0,Y 473.736,Z 630.762,A -85,B 0,C 180,E1 -7292.551,E2 -7292.551} C_VEL
LIN {X 0,Y 473.693,Z 628.43,A -85,B 0,C 180,E1 -7294.255,E2 -7294.255} C_VEL
LIN {X 0,Y 473.782,Z 624.892,A -85,B 0,C 180,E1 -7295.96,E2 -7295.96} C_VEL
LIN {X 0,Y 473.911,Z 620.054,A -85,B 0,C 180,E1 -7297.67,E2 -7297.67} C_VEL
LIN {X 0,Y 474.111,Z 613.786,A -85,B 0,C 180,E1 -7299.385,E2 -7299.385} C_VEL
LIN {X 0,Y 474.521,Z 605.916,A -85,B 0,C 180,E1 -7301.101,E2 -7301.101} C_VEL
LIN {X 0,Y 474.903,Z 597.301,A -85,B 0,C 180,E1 -7302.646,E2 -7302.646} C_VEL
LIN {X 0,Y 475.446,Z 587.443,A -85,B 0,C 180,E1 -7304.117,E2 -7304.117} C_VEL
LIN {X 0,Y 476.052,Z 577.133,A -85,B 0,C 180,E1 -7305.411,E2 -7305.411} C_VEL
LIN {X 0,Y 476.858,Z 565.165,A -85,B 0,C 180,E1 -7306.668,E2 -7306.668} C_VEL
LIN {X 0,Y 477.627,Z 552.463,A -85,B 0,C 180,E1 -7307.778,E2 -7307.778} C_VEL
LIN {X 0,Y 478.466,Z 538.99,A -85,B 0,C 180,E1 -7308.742,E2 -7308.742} C_VEL
LIN {X 0,Y 479.237,Z 524.079,A -85,B 0,C 180,E1 -7309.6,E2 -7309.6} C_VEL
LIN {X 0,Y 479.954,Z 508.646,A -85,B 0,C 180,E1 -7310.277,E2 -7310.277} C_VEL
LIN {X 0,Y 480.514,Z 493.896,A -85,B 0,C 180,E1 -7310.746,E2 -7310.746} C_VEL
LIN {X 0,Y 480.82,Z 478.393,A -85,B 0,C 180,E1 -7311.068,E2 -7311.068} C_VEL
LIN {X 0,Y 482.383,Z 342.343,A -85,B 0,C 180,E1 -7313.164,E2 -7313.164} C_VEL
LIN {X 0,Y 477.985,Z 319.613,A -85,B 0,C 180,E1 -7313.773,E2 -7313.773} C_VEL
LIN {X 0,Y 479.034,Z 299.54,A -85,B 0,C 180,E1 -7316.689,E2 -7316.689} C_VEL
LIN {X 0,Y 478.588,Z 295.604,A -85,B 0,C 180,E1 -7317.305,E2 -7317.305} C_VEL
LIN {X 0,Y 475.198,Z 281.273,A -85,B 0,C 180,E1 -7319.699,E2 -7319.699} C_VEL
LIN {X 0,Y 474.648,Z 278.978,A -85,B 0,C 180,E1 -7320.104,E2 -7320.104} C_VEL
LIN {X 0,Y 474.616,Z 278.99,A -85,B 0,C 180,E1 -7323.222,E2 -7323.222} C_VEL
LIN {X 0,Y 474.581,Z 278.998,A -85,B 0,C 180,E1 -7326.324,E2 -7326.324} C_VEL
LIN {X 0,Y 474.601,Z 278.994,A -85,B 0,C 180,E1 -7329.643,E2 -7329.643} C_VEL
LIN {X 0,Y 474.568,Z 278.99,A -85,B 0,C 180,E1 -7332.939,E2 -7332.939} C_VEL
LIN {X 0,Y 474.601,Z 278.993,A -85,B 0,C 180,E1 -7335.893,E2 -7335.893} C_VEL
LIN {X 0,Y 474.6,Z 278.991,A -85,B 0,C 180,E1 -7339.044,E2 -7339.044} C_VEL
LIN {X 0,Y 474.588,Z 278.992,A -85,B 0,C 180,E1 -7341.706,E2 -7341.706} C_VEL
LIN {X 0,Y 474.608,Z 278.984,A -85,B 0,C 180,E1 -7344.723,E2 -7344.723} C_VEL
LIN {X 0,Y 474.625,Z 278.99,A -85,B 0,C 180,E1 -7347.786,E2 -7347.786} C_VEL
LIN {X 0,Y 474.599,Z 278.988,A -85,B 0,C 180,E1 -7350.889,E2 -7350.889} C_VEL
LIN {X 0,Y 474.577,Z 278.994,A -85,B 0,C 180,E1 -7353.622,E2 -7353.622} C_VEL
LIN {X 0,Y 474.631,Z 278.984,A -85,B 0,C 180,E1 -7356.641,E2 -7356.641} C_VEL
LIN {X 0,Y 474.647,Z 278.985,A -85,B 0,C 180,E1 -7360.088,E2 -7360.088} C_VEL
LIN {X 0,Y 474.622,Z 278.987,A -85,B 0,C 180,E1 -7362.772,E2 -7362.772} C_VEL
LIN {X 0,Y 474.639,Z 278.985,A -85,B 0,C 180,E1 -7365.42,E2 -7365.42} C_VEL
LIN {X 0,Y 474.686,Z 278.971,A -85,B 0,C 180,E1 -7368.036,E2 -7368.036} C_VEL
LIN {X 0,Y 474.654,Z 278.986,A -85,B 0,C 180,E1 -7371.484,E2 -7371.484} C_VEL
LIN {X 0,Y 474.73,Z 278.97,A -85,B 0,C 180,E1 -7374.051,E2 -7374.051} C_VEL
LIN {X 0,Y 474.836,Z 278.949,A -85,B 0,C 180,E1 -7377.454,E2 -7377.454} C_VEL
LIN {X 0,Y 474.867,Z 278.956,A -85,B 0,C 180,E1 -7379.999,E2 -7379.999} C_VEL
LIN {X 0,Y 474.869,Z 278.953,A -85,B 0,C 180,E1 -7382.543,E2 -7382.543} C_VEL
LIN {X 0,Y 474.705,Z 278.96,A -85,B 0,C 180,E1 -7385.947,E2 -7385.947} C_VEL
LIN {X 0,Y 474.659,Z 278.98,A -85,B 0,C 180,E1 -7389.372,E2 -7389.372} C_VEL
LIN {X 0,Y 474.691,Z 278.976,A -85,B 0,C 180,E1 -7392.274,E2 -7392.274} C_VEL
LIN {X 0,Y 474.668,Z 278.968,A -85,B 0,C 180,E1 -7395.765,E2 -7395.765} C_VEL
LIN {X 0,Y 474.647,Z 278.976,A -85,B 0,C 180,E1 -7399.009,E2 -7399.009} C_VEL
LIN {X 0,Y 474.575,Z 278.993,A -85,B 0,C 180,E1 -7401.728,E2 -7401.728} C_VEL
LIN {X 0,Y 474.612,Z 278.983,A -85,B 0,C 180,E1 -7404.493,E2 -7404.493} C_VEL
LIN {X 0,Y 474.585,Z 278.98,A -85,B 0,C 180,E1 -7407.325,E2 -7407.325} C_VEL
LIN {X 0,Y 474.582,Z 278.987,A -85,B 0,C 180,E1 -7410.23,E2 -7410.23} C_VEL
LIN {X 0,Y 474.6,Z 278.992,A -85,B 0,C 180,E1 -7413.221,E2 -7413.221} C_VEL
LIN {X 0,Y 474.568,Z 278.98,A -85,B 0,C 180,E1 -7416.323,E2 -7416.323} C_VEL
LIN {X 0,Y 474.607,Z 278.989,A -85,B 0,C 180,E1 -7419.547,E2 -7419.547} C_VEL
LIN {X 0,Y 474.572,Z 278.991,A -85,B 0,C 180,E1 -7422.231,E2 -7422.231} C_VEL
LIN {X 0,Y 474.599,Z 278.983,A -85,B 0,C 180,E1 -7425.297,E2 -7425.297} C_VEL
LIN {X 0,Y 474.598,Z 278.988,A -85,B 0,C 180,E1 -7428.213,E2 -7428.213} C_VEL
LIN {X 0,Y 474.594,Z 278.986,A -85,B 0,C 180,E1 -7431.542,E2 -7431.542} C_VEL
LIN {X 0,Y 474.606,Z 278.988,A -85,B 0,C 180,E1 -7434.725,E2 -7434.725} C_VEL
